LIN {X 0,Y 355.069,Z 437.822,A -85,B 0,C 180,E1 -13382.962,E2 -13382.962} C_VEL
LIN {X 0,Y 354.55,Z 443.957,A -85,B 0,C 180,E1 -13386.644,E2 -13386.644} C_VEL
LIN {X 0,Y 354.327,Z 447.213,A -85,B 0,C 180,E1 -13388.544,E2 -13388.544} C_VEL
LIN {X 0,Y 357.927,Z 462.042,A -85,B 0,C 180,E1 -13389.4,E2 -13389.4} C_VEL
LIN {X 0,Y 360.061,Z 473.49,A -85,B 0,C 180,E1 -13390.214,E2 -13390.214} C_VEL
LIN {X 0,Y 361.071,Z 484.49,A -85,B 0,C 180,E1 -13391.12,E2 -13391.12} C_VEL
LIN {X 0,Y 360.323,Z 493.852,A -85,B 0,C 180,E1 -13391.963,E2 -13391.963} C_VEL
LIN {X 0,Y 358.816,Z 505.238,A -85,B 0,C 180,E1 -13393.208,E2 -13393.208} C_VEL
LIN {X 0,Y 357.676,Z 514.692,A -85,B 0,C 180,E1 -13394.514,E2 -13394.514} C_VEL
LIN {X 0,Y 356.51,Z 523.583,A -85,B 0,C 180,E1 -13396.026,E2 -13396.026} C_VEL
LIN {X 0,Y 355.306,Z 531.692,A -85,B 0,C 180,E1 -13397.723,E2 -13397.723} C_VEL
LIN {X 0,Y 354.632,Z 537.229,A -85,B 0,C 180,E1 -13399.148,E2 -13399.148} C_VEL
LIN {X 0,Y 353.992,Z 542.659,A -85,B 0,C 180,E1 -13400.861,E2 -13400.861} C_VEL
LIN {X 0,Y 353.532,Z 546.923,A -85,B 0,C 180,E1 -13402.576,E2 -13402.576} C_VEL
LIN {X 0,Y 353.311,Z 550.14,A -85,B 0,C 180,E1 -13404.292,E2 -13404.292} C_VEL
LIN {X 0,Y 353.267,Z 551.75,A -85,B 0,C 180,E1 -13405.436,E2 -13405.436} C_VEL
LIN {X 0,Y 353.22,Z 552.959,A -85,B 0,C 180,E1 -13406.578,E2 -13406.578} C_VEL
LIN {X 0,Y 353.216,Z 554.108,A -85,B 0,C 180,E1 -13408.86,E2 -13408.86} C_VEL
LIN {X 0,Y 353.263,Z 554.103,A -85,B 0,C 180,E1 -13410,E2 -13410} C_VEL
LIN {X 0,Y 353.222,Z 553.708,A -85,B 0,C 180,E1 -13411.14,E2 -13411.14} C_VEL
LIN {X 0,Y 353.186,Z 552.882,A -85,B 0,C 180,E1 -13412.281,E2 -13412.281} C_VEL
LIN {X 0,Y 353.225,Z 551.643,A -85,B 0,C 180,E1 -13413.422,E2 -13413.422} C_VEL
LIN {X 0,Y 353.253,Z 548.999,A -85,B 0,C 180,E1 -13415.136,E2 -13415.136} C_VEL
LIN {X 0,Y 353.417,Z 545.326,A -85,B 0,C 180,E1 -13416.852,E2 -13416.852} C_VEL
LIN {X 0,Y 353.731,Z 540.524,A -85,B 0,C 180,E1 -13418.569,E2 -13418.569} C_VEL
LIN {X 0,Y 354.312,Z 533.318,A -85,B 0,C 180,E1 -13420.572,E2 -13420.572} C_VEL
LIN {X 0,Y 355.049,Z 525.43,A -85,B 0,C 180,E1 -13422.285,E2 -13422.285} C_VEL
LIN {X 0,Y 355.823,Z 517.369,A -85,B 0,C 180,E1 -13423.71,E2 -13423.71} C_VEL
LIN {X 0,Y 356.72,Z 507.617,A -85,B 0,C 180,E1 -13425.119,E2 -13425.119} C_VEL
LIN {X 0,Y 357.759,Z 496.542,A -85,B 0,C 180,E1 -13426.402,E2 -13426.402} C_VEL
LIN {X 0,Y 358.683,Z 485.774,A -85,B 0,C 180,E1 -13427.385,E2 -13427.385} C_VEL
LIN {X 0,Y 358.573,Z 480.17,A -85,B 0,C 180,E1 -13427.833,E2 -13427.833} C_VEL
LIN {X 0,Y 357.135,Z 467.764,A -85,B 0,C 180,E1 -13428.691,E2 -13428.691} C_VEL
LIN {X 0,Y 355.076,Z 454.636,A -85,B 0,C 180,E1 -13429.383,E2 -13429.383} C_VEL
LIN {X 0,Y 353.874,Z 447.574,A -85,B 0,C 180,E1 -13429.689,E2 -13429.689} C_VEL
LIN {X 0,Y 354.228,Z 442.075,A -85,B 0,C 180,E1 -13432.76,E2 -13432.76} C_VEL
LIN {X 0,Y 354.602,Z 436.609,A -85,B 0,C 180,E1 -13435.85,E2 -13435.85} C_VEL
LIN {X 0,Y 355.244,Z 428.947,A -85,B 0,C 180,E1 -13440.296,E2 -13440.296} C_VEL
LIN {X 0,Y 355.742,Z 423.445,A -85,B 0,C 180,E1 -13443.583,E2 -13443.583} C_VEL
LIN {X 0,Y 355.998,Z 419.022,A -85,B 0,C 180,E1 -13446.316,E2 -13446.316} C_VEL
LIN {X 0,Y 355.661,Z 415.659,A -85,B 0,C 180,E1 -13448.494,E2 -13448.494} C_VEL
LIN {X 0,Y 354.899,Z 411.28,A -85,B 0,C 180,E1 -13451.56,E2 -13451.56} C_VEL
LIN {X 0,Y 354.812,Z 411.288,A -85,B 0,C 180,E1 -13455.484,E2 -13455.484} C_VEL
LIN {X 0,Y 354.785,Z 411.293,A -85,B 0,C 180,E1 -13459.178,E2 -13459.178} C_VEL
LIN {X 0,Y 354.804,Z 411.287,A -85,B 0,C 180,E1 -13462.401,E2 -13462.401} C_VEL
LIN {X 0,Y 354.808,Z 411.291,A -85,B 0,C 180,E1 -13464.94,E2 -13464.94} C_VEL
LIN {X 0,Y 354.788,Z 411.29,A -85,B 0,C 180,E1 -13468.404,E2 -13468.404} C_VEL
LIN {X 0,Y 354.848,Z 411.281,A -85,B 0,C 180,E1 -13471.619,E2 -13471.619} C_VEL
LIN {X 0,Y 354.893,Z 411.276,A -85,B 0,C 180,E1 -13474.172,E2 -13474.172} C_VEL
LIN {X 0,Y 354.828,Z 411.283,A -85,B 0,C 180,E1 -13477.893,E2 -13477.893} C_VEL
LIN {X 0,Y 354.915,Z 411.273,A -85,B 0,C 180,E1 -13481.891,E2 -13481.891} C_VEL
LIN {X 0,Y 354.935,Z 411.271,A -85,B 0,C 180,E1 -13485.981,E2 -13485.981} C_VEL
LIN {X 0,Y 354.97,Z 411.266,A -85,B 0,C 180,E1 -13489.735,E2 -13489.735} C_VEL
LIN {X 0,Y 355.121,Z 411.249,A -85,B 0,C 180,E1 -13492.037,E2 -13492.037} C_VEL
LIN {X 0,Y 355.089,Z 411.256,A -85,B 0,C 180,E1 -13494.32,E2 -13494.32} C_VEL
LIN {X 0,Y 355.239,Z 411.233,A -85,B 0,C 180,E1 -13497.732,E2 -13497.732} C_VEL
LIN {X 0,Y 355.391,Z 411.216,A -85,B 0,C 180,E1 -13500,E2 -13500} C_VEL
LIN {X 0,Y 355.239,Z 411.237,A -85,B 0,C 180,E1 -13502.267,E2 -13502.267} C_VEL
LIN {X 0,Y 355.13,Z 411.247,A -85,B 0,C 180,E1 -13506.819,E2 -13506.819} C_VEL
LIN {X 0,Y 355.008,Z 411.261,A -85,B 0,C 180,E1 -13509.112,E2 -13509.112} C_VEL
LIN {X 0,Y 354.916,Z 411.274,A -85,B 0,C 180,E1 -13512.581,E2 -13512.581} C_VEL
LIN {X 0,Y 354.882,Z 411.282,A -85,B 0,C 180,E1 -13516.096,E2 -13516.096} C_VEL
LIN {X 0,Y 354.896,Z 411.277,A -85,B 0,C 180,E1 -13518.472,E2 -13518.472} C_VEL
LIN {X 0,Y 354.827,Z 411.288,A -85,B 0,C 180,E1 -13522.106,E2 -13522.106} C_VEL
LIN {X 0,Y 354.892,Z 411.28,A -85,B 0,C 180,E1 -13525.828,E2 -13525.828} C_VEL
LIN {X 0,Y 354.848,Z 411.285,A -85,B 0,C 180,E1 -13529.679,E2 -13529.679} C_VEL
LIN {X 0,Y 354.824,Z 411.289,A -85,B 0,C 180,E1 -13533.683,E2 -13533.683} C_VEL
LIN {X 0,Y 354.796,Z 411.287,A -85,B 0,C 180,E1 -13536.46,E2 -13536.46} C_VEL
LIN {X 0,Y 354.818,Z 411.288,A -85,B 0,C 180,E1 -13539.424,E2 -13539.424} C_VEL
LIN {X 0,Y 354.837,Z 411.282,A -85,B 0,C 180,E1 -13542.877,E2 -13542.877} C_VEL
LIN {X 0,Y 354.861,Z 411.28,A -85,B 0,C 180,E1 -13546.12,E2 -13546.12} C_VEL
LIN {X 0,Y 354.852,Z 411.283,A -85,B 0,C 180,E1 -13549.189,E2 -13549.189} C_VEL
LIN {X 0,Y 354.806,Z 411.285,A -85,B 0,C 180,E1 -13552.403,E2 -13552.403} C_VEL
LIN {X 0,Y 354.809,Z 411.287,A -85,B 0,C 180,E1 -13554.942,E2 -13554.942} C_VEL
LIN {X 0,Y 354.79,Z 411.288,A -85,B 0,C 180,E1 -13558.406,E2 -13558.406} C_VEL
LIN {X 0,Y 354.849,Z 411.283,A -85,B 0,C 180,E1 -13561.62,E2 -13561.62} C_VEL
LIN {X 0,Y 354.896,Z 411.274,A -85,B 0,C 180,E1 -13564.173,E2 -13564.173} C_VEL
LIN {X 0,Y 354.792,Z 411.289,A -85,B 0,C 180,E1 -13566.661,E2 -13566.661} C_VEL
LIN {X 0,Y 354.679,Z 411.364,A -85,B 0,C 180,E1 -13569.257,E2 -13569.257} C_VEL
LIN {X 0,Y 354.506,Z 415.32,A -85,B 0,C 180,E1 -13572.701,E2 -13572.701} C_VEL
LIN {X 0,Y 354.361,Z 419.603,A -85,B 0,C 180,E1 -13576.363,E2 -13576.363} C_VEL
LIN {X 0,Y 354.088,Z 423.661,A -85,B 0,C 180,E1 -13579.71,E2 -13579.71} C_VEL
LIN {X 0,Y 354.096,Z 427.875,A -85,B 0,C 180,E1 -13583.161,E2 -13583.161} C_VEL
LIN {X 0,Y 353.953,Z 429.544,A -85,B 0,C 180,E1 -13584.446,E2 -13584.446} C_VEL
LIN {X 0,Y 356.736,Z 442.632,A -85,B 0,C 180,E1 -13585.073,E2 -13585.073} C_VEL
LIN {X 0,Y 358.816,Z 454.707,A -85,B 0,C 180,E1 -13585.847,E2 -13585.847} C_VEL
LIN {X 0,Y 359.504,Z 461.1,A -85,B 0,C 180,E1 -13586.328,E2 -13586.328} C_VEL
LIN {X 0,Y 358.588,Z 472.632,A -85,B 0,C 180,E1 -13587.29,E2 -13587.29} C_VEL
LIN {X 0,Y 357.635,Z 483.505,A -85,B 0,C 180,E1 -13588.452,E2 -13588.452} C_VEL
LIN {X 0,Y 356.672,Z 493.088,A -85,B 0,C 180,E1 -13589.718,E2 -13589.718} C_VEL
LIN {X 0,Y 355.798,Z 501.822,A -85,B 0,C 180,E1 -13591.132,E2 -13591.132} C_VEL
LIN {X 0,Y 354.892,Z 510.326,A -85,B 0,C 180,E1 -13592.838,E2 -13592.838} C_VEL
LIN {X 0,Y 354.214,Z 517.147,A -85,B 0,C 180,E1 -13594.552,E2 -13594.552} C_VEL
LIN {X 0,Y 353.84,Z 522.956,A -85,B 0,C 180,E1 -13596.401,E2 -13596.401} C_VEL
LIN {X 0,Y 353.541,Z 526.863,A -85,B 0,C 180,E1 -13597.999,E2 -13597.999} C_VEL
LIN {X 0,Y 353.345,Z 529.138,A -85,B 0,C 180,E1 -13599.156,E2 -13599.156} C_VEL
LIN {X 0,Y 353.202,Z 530.929,A -85,B 0,C 180,E1 -13600.316,E2 -13600.316} C_VEL
LIN {X 0,Y 353.163,Z 532.281,A -85,B 0,C 180,E1 -13601.479,E2 -13601.479} C_VEL
LIN {X 0,Y 353.134,Z 533.337,A -85,B 0,C 180,E1 -13602.79,E2 -13602.79} C_VEL
LIN {X 0,Y 353.028,Z 533.879,A -85,B 0,C 180,E1 -13604.999,E2 -13604.999} C_VEL
LIN {X 0,Y 353.191,Z 532.951,A -85,B 0,C 180,E1 -13607.229,E2 -13607.229} C_VEL
LIN {X 0,Y 353.364,Z 531.684,A -85,B 0,C 180,E1 -13608.555,E2 -13608.555} C_VEL
LIN {X 0,Y 353.729,Z 529.087,A -85,B 0,C 180,E1 -13610.346,E2 -13610.346} C_VEL
LIN {X 0,Y 354.177,Z 525.384,A -85,B 0,C 180,E1 -13612.149,E2 -13612.149} C_VEL
LIN {X 0,Y 354.83,Z 520.648,A -85,B 0,C 180,E1 -13613.893,E2 -13613.893} C_VEL
LIN {X 0,Y 355.718,Z 514.138,A -85,B 0,C 180,E1 -13615.763,E2 -13615.763} C_VEL
LIN {X 0,Y 356.686,Z 507.497,A -85,B 0,C 180,E1 -13617.291,E2 -13617.291} C_VEL
LIN {X 0,Y 357.752,Z 499.676,A -85,B 0,C 180,E1 -13618.77,E2 -13618.77} C_VEL
LIN {X 0,Y 359.127,Z 489.929,A -85,B 0,C 180,E1 -13620.259,E2 -13620.259} C_VEL
LIN {X 0,Y 360.487,Z 478.928,A -85,B 0,C 180,E1 -13621.597,E2 -13621.597} C_VEL
LIN {X 0,Y 361.665,Z 468.228,A -85,B 0,C 180,E1 -13622.632,E2 -13622.632} C_VEL
LIN {X 0,Y 362.126,Z 461.499,A -85,B 0,C 180,E1 -13623.181,E2 -13623.181} C_VEL
LIN {X 0,Y 359.869,Z 449.843,A -85,B 0,C 180,E1 -13624.152,E2 -13624.152} C_VEL
LIN {X 0,Y 356.437,Z 437.583,A -85,B 0,C 180,E1 -13625.027,E2 -13625.027} C_VEL
LIN {X 0,Y 353.983,Z 429.889,A -85,B 0,C 180,E1 -13625.51,E2 -13625.51} C_VEL
LIN {X 0,Y 354.281,Z 425.752,A -85,B 0,C 180,E1 -13629.109,E2 -13629.109} C_VEL
LIN {X 0,Y 353.723,Z 424.789,A -85,B 0,C 180,E1 -13630.046,E2 -13630.046} C_VEL
LIN {X 0,Y 350.983,Z 423.48,A -85,B 0,C 180,E1 -13631.58,E2 -13631.58} C_VEL
LIN {X 0,Y 348.634,Z 422.481,A -85,B 0,C 180,E1 -13632.822,E2 -13632.822} C_VEL
LIN {X 0,Y 347.655,Z 421.607,A -85,B 0,C 180,E1 -13633.779,E2 -13633.779} C_VEL
LIN {X 0,Y 347.595,Z 421.276,A -85,B 0,C 180,E1 -13634.102,E2 -13634.102} C_VEL
LIN {X 0,Y 347.873,Z 418.606,A -85,B 0,C 180,E1 -13636.66,E2 -13636.66} C_VEL
LIN {X 0,Y 348.008,Z 415.552,A -85,B 0,C 180,E1 -13639.742,E2 -13639.742} C_VEL
LIN {X 0,Y 347.833,Z 412.784,A -85,B 0,C 180,E1 -13642.688,E2 -13642.688} C_VEL
LIN {X 0,Y 347.783,Z 412.171,A -85,B 0,C 180,E1 -13644.124,E2 -13644.124} C_VEL
LIN {X 0,Y 347.749,Z 412.172,A -85,B 0,C 180,E1 -13648.082,E2 -13648.082} C_VEL
LIN {X 0,Y 347.802,Z 412.162,A -85,B 0,C 180,E1 -13650.99,E2 -13650.99} C_VEL
LIN {X 0,Y 347.827,Z 412.159,A -85,B 0,C 180,E1 -13653.608,E2 -13653.608} C_VEL
LIN {X 0,Y 347.781,Z 412.164,A -85,B 0,C 180,E1 -13656.162,E2 -13656.162} C_VEL
LIN {X 0,Y 347.806,Z 412.161,A -85,B 0,C 180,E1 -13659.909,E2 -13659.909} C_VEL
LIN {X 0,Y 347.861,Z 412.153,A -85,B 0,C 180,E1 -13662.359,E2 -13662.359} C_VEL
LIN {X 0,Y 347.892,Z 412.147,A -85,B 0,C 180,E1 -13665.971,E2 -13665.971} C_VEL
LIN {X 0,Y 347.923,Z 412.144,A -85,B 0,C 180,E1 -13669.526,E2 -13669.526} C_VEL
LIN {X 0,Y 348.069,Z 412.129,A -85,B 0,C 180,E1 -13671.875,E2 -13671.875} C_VEL
LIN {X 0,Y 348.062,Z 412.129,A -85,B 0,C 180,E1 -13674.206,E2 -13674.206} C_VEL
LIN {X 0,Y 348.203,Z 412.111,A -85,B 0,C 180,E1 -13677.687,E2 -13677.687} C_VEL
LIN {X 0,Y 348.341,Z 412.095,A -85,B 0,C 180,E1 -13680,E2 -13680} C_VEL
LIN {X 0,Y 348.203,Z 412.113,A -85,B 0,C 180,E1 -13682.314,E2 -13682.314} C_VEL
LIN {X 0,Y 348.089,Z 412.122,A -85,B 0,C 180,E1 -13686.958,E2 -13686.958} C_VEL
LIN {X 0,Y 347.928,Z 412.146,A -85,B 0,C 180,E1 -13690.475,E2 -13690.475} C_VEL
LIN {X 0,Y 347.894,Z 412.15,A -85,B 0,C 180,E1 -13694.15,E2 -13694.15} C_VEL
LIN {X 0,Y 347.887,Z 412.153,A -85,B 0,C 180,E1 -13698.291,E2 -13698.291} C_VEL
LIN {X 0,Y 347.785,Z 412.167,A -85,B 0,C 180,E1 -13701.635,E2 -13701.635} C_VEL
LIN {X 0,Y 347.809,Z 412.164,A -85,B 0,C 180,E1 -13705.109,E2 -13705.109} C_VEL
LIN {X 0,Y 347.809,Z 412.164,A -85,B 0,C 180,E1 -13707.694,E2 -13707.694} C_VEL
LIN {X 0,Y 347.761,Z 412.168,A -85,B 0,C 180,E1 -13710.347,E2 -13710.347} C_VEL
LIN {X 0,Y 347.742,Z 412.169,A -85,B 0,C 180,E1 -13714.465,E2 -13714.465} C_VEL
LIN {X 0,Y 347.772,Z 412.158,A -85,B 0,C 180,E1 -13717.989,E2 -13717.989} C_VEL
LIN {X 0,Y 347.749,Z 412.17,A -85,B 0,C 180,E1 -13721.831,E2 -13721.831} C_VEL
LIN {X 0,Y 347.76,Z 412.322,A -85,B 0,C 180,E1 -13723.803,E2 -13723.803} C_VEL
LIN {X 0,Y 348.361,Z 415.62,A -85,B 0,C 180,E1 -13726.692,E2 -13726.692} C_VEL
LIN {X 0,Y 349.056,Z 419.568,A -85,B 0,C 180,E1 -13729.917,E2 -13729.917} C_VEL
LIN {X 0,Y 349.61,Z 424.356,A -85,B 0,C 180,E1 -13733.524,E2 -13733.524} C_VEL
LIN {X 0,Y 349.289,Z 428.522,A -85,B 0,C 180,E1 -13736.405,E2 -13736.405} C_VEL
LIN {X 0,Y 348.599,Z 434.182,A -85,B 0,C 180,E1 -13740.102,E2 -13740.102} C_VEL
LIN {X 0,Y 347.818,Z 440.809,A -85,B 0,C 180,E1 -13744.251,E2 -13744.251} C_VEL
LIN {X 0,Y 347.321,Z 447.037,A -85,B 0,C 180,E1 -13748.016,E2 -13748.016} C_VEL
LIN {X 0,Y 350.748,Z 460.4,A -85,B 0,C 180,E1 -13748.797,E2 -13748.797} C_VEL
LIN {X 0,Y 353.117,Z 472.607,A -85,B 0,C 180,E1 -13749.679,E2 -13749.679} C_VEL
LIN {X 0,Y 354.288,Z 483.47,A -85,B 0,C 180,E1 -13750.594,E2 -13750.594} C_VEL
LIN {X 0,Y 354.153,Z 489.992,A -85,B 0,C 180,E1 -13751.188,E2 -13751.188} C_VEL
LIN {X 0,Y 352.75,Z 500.954,A -85,B 0,C 180,E1 -13752.312,E2 -13752.312} C_VEL
LIN {X 0,Y 351.477,Z 509.868,A -85,B 0,C 180,E1 -13753.445,E2 -13753.445} C_VEL
LIN {X 0,Y 350.311,Z 519.035,A -85,B 0,C 180,E1 -13754.882,E2 -13754.882} C_VEL
LIN {X 0,Y 348.992,Z 527.977,A -85,B 0,C 180,E1 -13756.61,E2 -13756.61} C_VEL
LIN {X 0,Y 347.862,Z 535.203,A -85,B 0,C 180,E1 -13758.344,E2 -13758.344} C_VEL
LIN {X 0,Y 347.143,Z 541.01,A -85,B 0,C 180,E1 -13760.091,E2 -13760.091} C_VEL
LIN {X 0,Y 346.633,Z 545.603,A -85,B 0,C 180,E1 -13761.841,E2 -13761.841} C_VEL
LIN {X 0,Y 346.243,Z 549.837,A -85,B 0,C 180,E1 -13764.044,E2 -13764.044} C_VEL
LIN {X 0,Y 346.167,Z 551.63,A -85,B 0,C 180,E1 -13765.342,E2 -13765.342} C_VEL
LIN {X 0,Y 346.143,Z 552.81,A -85,B 0,C 180,E1 -13766.508,E2 -13766.508} C_VEL
LIN {X 0,Y 346.116,Z 553.913,A -85,B 0,C 180,E1 -13768.836,E2 -13768.836} C_VEL
LIN {X 0,Y 346.166,Z 553.888,A -85,B 0,C 180,E1 -13770,E2 -13770} C_VEL
LIN {X 0,Y 346.123,Z 553.469,A -85,B 0,C 180,E1 -13771.163,E2 -13771.163} C_VEL
LIN {X 0,Y 346.097,Z 552.611,A -85,B 0,C 180,E1 -13772.327,E2 -13772.327} C_VEL
LIN {X 0,Y 346.149,Z 551.353,A -85,B 0,C 180,E1 -13773.492,E2 -13773.492} C_VEL
LIN {X 0,Y 346.167,Z 548.283,A -85,B 0,C 180,E1 -13775.45,E2 -13775.45} C_VEL
LIN {X 0,Y 346.449,Z 543.491,A -85,B 0,C 180,E1 -13777.577,E2 -13777.577} C_VEL
LIN {X 0,Y 346.879,Z 537.209,A -85,B 0,C 180,E1 -13779.622,E2 -13779.622} C_VEL
LIN {X 0,Y 347.455,Z 530.358,A -85,B 0,C 180,E1 -13781.374,E2 -13781.374} C_VEL
LIN {X 0,Y 348.432,Z 521.825,A -85,B 0,C 180,E1 -13783.115,E2 -13783.115} C_VEL
LIN {X 0,Y 349.341,Z 513.023,A -85,B 0,C 180,E1 -13784.564,E2 -13784.564} C_VEL
LIN {X 0,Y 350.126,Z 503.701,A -85,B 0,C 180,E1 -13785.827,E2 -13785.827} C_VEL
LIN {X 0,Y 351.177,Z 492.787,A -85,B 0,C 180,E1 -13787.018,E2 -13787.018} C_VEL
LIN {X 0,Y 351.848,Z 482.92,A -85,B 0,C 180,E1 -13787.884,E2 -13787.884} C_VEL
LIN {X 0,Y 350.499,Z 470.9,A -85,B 0,C 180,E1 -13788.795,E2 -13788.795} C_VEL
LIN {X 0,Y 348.564,Z 457.645,A -85,B 0,C 180,E1 -13789.555,E2 -13789.555} C_VEL
LIN {X 0,Y 346.846,Z 447.401,A -85,B 0,C 180,E1 -13790.019,E2 -13790.019} C_VEL
LIN {X 0,Y 347.206,Z 441.747,A -85,B 0,C 180,E1 -13793.247,E2 -13793.247} C_VEL
LIN {X 0,Y 347.573,Z 436.299,A -85,B 0,C 180,E1 -13796.413,E2 -13796.413} C_VEL
LIN {X 0,Y 348.193,Z 429.725,A -85,B 0,C 180,E1 -13800.304,E2 -13800.304} C_VEL
LIN {X 0,Y 348.598,Z 425.337,A -85,B 0,C 180,E1 -13802.979,E2 -13802.979} C_VEL
LIN {X 0,Y 348.952,Z 420.922,A -85,B 0,C 180,E1 -13805.736,E2 -13805.736} C_VEL
LIN {X 0,Y 348.719,Z 417.179,A -85,B 0,C 180,E1 -13808.187,E2 -13808.187} C_VEL
LIN {X 0,Y 347.838,Z 412.16,A -85,B 0,C 180,E1 -13811.816,E2 -13811.816} C_VEL
LIN {X 0,Y 347.793,Z 412.164,A -85,B 0,C 180,E1 -13815.011,E2 -13815.011} C_VEL
LIN {X 0,Y 347.747,Z 412.166,A -85,B 0,C 180,E1 -13818.396,E2 -13818.396} C_VEL
LIN {X 0,Y 347.77,Z 412.162,A -85,B 0,C 180,E1 -13822.01,E2 -13822.01} C_VEL
LIN {X 0,Y 347.74,Z 412.167,A -85,B 0,C 180,E1 -13825.535,E2 -13825.535} C_VEL
LIN {X 0,Y 347.759,Z 412.164,A -85,B 0,C 180,E1 -13829.653,E2 -13829.653} C_VEL
LIN {X 0,Y 347.847,Z 412.158,A -85,B 0,C 180,E1 -13832.744,E2 -13832.744} C_VEL
LIN {X 0,Y 347.782,Z 412.162,A -85,B 0,C 180,E1 -13836.161,E2 -13836.161} C_VEL
LIN {X 0,Y 347.806,Z 412.158,A -85,B 0,C 180,E1 -13839.909,E2 -13839.909} C_VEL
LIN {X 0,Y 347.859,Z 412.154,A -85,B 0,C 180,E1 -13842.359,E2 -13842.359} C_VEL
LIN {X 0,Y 347.89,Z 412.148,A -85,B 0,C 180,E1 -13845.97,E2 -13845.97} C_VEL
LIN {X 0,Y 347.921,Z 412.143,A -85,B 0,C 180,E1 -13849.525,E2 -13849.525} C_VEL
LIN {X 0,Y 348.103,Z 412.122,A -85,B 0,C 180,E1 -13853.042,E2 -13853.042} C_VEL
LIN {X 0,Y 348.201,Z 412.109,A -85,B 0,C 180,E1 -13857.686,E2 -13857.686} C_VEL
LIN {X 0,Y 348.361,Z 412.091,A -85,B 0,C 180,E1 -13860,E2 -13860} C_VEL
LIN {X 0,Y 348.201,Z 412.114,A -85,B 0,C 180,E1 -13862.313,E2 -13862.313} C_VEL
LIN {X 0,Y 348.098,Z 412.122,A -85,B 0,C 180,E1 -13866.958,E2 -13866.958} C_VEL
LIN {X 0,Y 347.96,Z 412.139,A -85,B 0,C 180,E1 -13869.299,E2 -13869.299} C_VEL
LIN {X 0,Y 347.884,Z 412.148,A -85,B 0,C 180,E1 -13872.839,E2 -13872.839} C_VEL
LIN {X 0,Y 347.832,Z 412.157,A -85,B 0,C 180,E1 -13876.432,E2 -13876.432} C_VEL
LIN {X 0,Y 347.845,Z 412.153,A -85,B 0,C 180,E1 -13878.861,E2 -13878.861} C_VEL
LIN {X 0,Y 347.767,Z 412.163,A -85,B 0,C 180,E1 -13882.58,E2 -13882.58} C_VEL
LIN {X 0,Y 347.805,Z 412.158,A -85,B 0,C 180,E1 -13885.109,E2 -13885.109} C_VEL
LIN {X 0,Y 347.805,Z 412.162,A -85,B 0,C 180,E1 -13887.694,E2 -13887.694} C_VEL
LIN {X 0,Y 347.764,Z 412.164,A -85,B 0,C 180,E1 -13890.346,E2 -13890.346} C_VEL
LIN {X 0,Y 347.742,Z 412.169,A -85,B 0,C 180,E1 -13894.044,E2 -13894.044} C_VEL
LIN {X 0,Y 347.761,Z 412.166,A -85,B 0,C 180,E1 -13897.321,E2 -13897.321} C_VEL
LIN {X 0,Y 347.788,Z 412.161,A -85,B 0,C 180,E1 -13900.289,E2 -13900.289} C_VEL
LIN {X 0,Y 347.814,Z 412.161,A -85,B 0,C 180,E1 -13903.394,E2 -13903.394} C_VEL
LIN {X 0,Y 347.813,Z 412.157,A -85,B 0,C 180,E1 -13906.671,E2 -13906.671} C_VEL
LIN {X 0,Y 347.782,Z 412.161,A -85,B 0,C 180,E1 -13910.166,E2 -13910.166} C_VEL
LIN {X 0,Y 347.786,Z 412.16,A -85,B 0,C 180,E1 -13914.126,E2 -13914.126} C_VEL
LIN {X 0,Y 347.735,Z 412.167,A -85,B 0,C 180,E1 -13918.087,E2 -13918.087} C_VEL
LIN {X 0,Y 347.803,Z 412.161,A -85,B 0,C 180,E1 -13920.991,E2 -13920.991} C_VEL
LIN {X 0,Y 347.829,Z 412.157,A -85,B 0,C 180,E1 -13923.608,E2 -13923.608} C_VEL
LIN {X 0,Y 347.768,Z 412.162,A -85,B 0,C 180,E1 -13926.161,E2 -13926.161} C_VEL
LIN {X 0,Y 347.624,Z 412.286,A -85,B 0,C 180,E1 -13929.281,E2 -13929.281} C_VEL
LIN {X 0,Y 347.473,Z 415.723,A -85,B 0,C 180,E1 -13932.339,E2 -13932.339} C_VEL
LIN {X 0,Y 347.303,Z 420.221,A -85,B 0,C 180,E1 -13936.246,E2 -13936.246} C_VEL
LIN {X 0,Y 347.002,Z 425.498,A -85,B 0,C 180,E1 -13940.676,E2 -13940.676} C_VEL
LIN {X 0,Y 346.978,Z 429.068,A -85,B 0,C 180,E1 -13943.604,E2 -13943.604} C_VEL
LIN {X 0,Y 346.92,Z 429.764,A -85,B 0,C 180,E1 -13944.114,E2 -13944.114} C_VEL
LIN {X 0,Y 349.778,Z 443.169,A -85,B 0,C 180,E1 -13944.777,E2 -13944.777} C_VEL
LIN {X 0,Y 351.789,Z 455.127,A -85,B 0,C 180,E1 -13945.56,E2 -13945.56} C_VEL
LIN {X 0,Y 352.642,Z 460.723,A -85,B 0,C 180,E1 -13946,E2 -13946} C_VEL
LIN {X 0,Y 351.729,Z 472.529,A -85,B 0,C 180,E1 -13946.993,E2 -13946.993} C_VEL
LIN {X 0,Y 350.665,Z 484.284,A -85,B 0,C 180,E1 -13948.278,E2 -13948.278} C_VEL
LIN {X 0,Y 349.573,Z 494.739,A -85,B 0,C 180,E1 -13949.712,E2 -13949.712} C_VEL
LIN {X 0,Y 348.675,Z 503.194,A -85,B 0,C 180,E1 -13951.155,E2 -13951.155} C_VEL
LIN {X 0,Y 347.752,Z 511.456,A -85,B 0,C 180,E1 -13952.896,E2 -13952.896} C_VEL
LIN {X 0,Y 347.096,Z 518.107,A -85,B 0,C 180,E1 -13954.646,E2 -13954.646} C_VEL
LIN {X 0,Y 346.75,Z 523.324,A -85,B 0,C 180,E1 -13956.373,E2 -13956.373} C_VEL
LIN {X 0,Y 346.439,Z 527.536,A -85,B 0,C 180,E1 -13958.164,E2 -13958.164} C_VEL
LIN {X 0,Y 346.222,Z 529.707,A -85,B 0,C 180,E1 -13959.346,E2 -13959.346} C_VEL
LIN {X 0,Y 346.098,Z 531.409,A -85,B 0,C 180,E1 -13960.53,E2 -13960.53} C_VEL
LIN {X 0,Y 346.05,Z 532.702,A -85,B 0,C 180,E1 -13961.718,E2 -13961.718} C_VEL
LIN {X 0,Y 346.047,Z 533.587,A -85,B 0,C 180,E1 -13962.909,E2 -13962.909} C_VEL
LIN {X 0,Y 345.951,Z 534.024,A -85,B 0,C 180,E1 -13964.11,E2 -13964.11} C_VEL
LIN {X 0,Y 345.94,Z 534.056,A -85,B 0,C 180,E1 -13965.314,E2 -13965.314} C_VEL
LIN {X 0,Y 346.146,Z 533.135,A -85,B 0,C 180,E1 -13967.395,E2 -13967.395} C_VEL
LIN {X 0,Y 346.331,Z 531.61,A -85,B 0,C 180,E1 -13968.946,E2 -13968.946} C_VEL
LIN {X 0,Y 346.599,Z 529.917,A -85,B 0,C 180,E1 -13970.164,E2 -13970.164} C_VEL
LIN {X 0,Y 347.054,Z 526.46,A -85,B 0,C 180,E1 -13972.001,E2 -13972.001} C_VEL
LIN {X 0,Y 347.735,Z 521.822,A -85,B 0,C 180,E1 -13973.842,E2 -13973.842} C_VEL
LIN {X 0,Y 348.626,Z 515.814,A -85,B 0,C 180,E1 -13975.685,E2 -13975.685} C_VEL
LIN {X 0,Y 349.777,Z 508.192,A -85,B 0,C 180,E1 -13977.525,E2 -13977.525} C_VEL
LIN {X 0,Y 350.932,Z 500.341,A -85,B 0,C 180,E1 -13979.054,E2 -13979.054} C_VEL
LIN {X 0,Y 352.325,Z 490.876,A -85,B 0,C 180,E1 -13980.552,E2 -13980.552} C_VEL
LIN {X 0,Y 353.652,Z 481.234,A -85,B 0,C 180,E1 -13981.777,E2 -13981.777} C_VEL
LIN {X 0,Y 354.812,Z 471.114,A -85,B 0,C 180,E1 -13982.824,E2 -13982.824} C_VEL
LIN {X 0,Y 355.511,Z 462.976,A -85,B 0,C 180,E1 -13983.525,E2 -13983.525} C_VEL
LIN {X 0,Y 353.281,Z 451.251,A -85,B 0,C 180,E1 -13984.55,E2 -13984.55} C_VEL
LIN {X 0,Y 349.669,Z 438.455,A -85,B 0,C 180,E1 -13985.512,E2 -13985.512} C_VEL
LIN {X 0,Y 346.959,Z 430.125,A -85,B 0,C 180,E1 -13986.054,E2 -13986.054} C_VEL
LIN {X 0,Y 347.229,Z 426.626,A -85,B 0,C 180,E1 -13989.145,E2 -13989.145} C_VEL
LIN {X 0,Y 347.496,Z 423.649,A -85,B 0,C 180,E1 -13991.867,E2 -13991.867} C_VEL
LIN {X 0,Y 347.595,Z 421.276,A -85,B 0,C 180,E1 -13994.102,E2 -13994.102} C_VEL
LIN {X 0,Y 347.009,Z 420.369,A -85,B 0,C 180,E1 -13995.059,E2 -13995.059} C_VEL
LIN {X 0,Y 344.308,Z 419.191,A -85,B 0,C 180,E1 -13996.629,E2 -13996.629} C_VEL
LIN {X 0,Y 342.007,Z 418.295,A -85,B 0,C 180,E1 -13997.901,E2 -13997.901} C_VEL
LIN {X 0,Y 341.039,Z 417.498,A -85,B 0,C 180,E1 -13998.879,E2 -13998.879} C_VEL
LIN {X 0,Y 340.971,Z 417.189,A -85,B 0,C 180,E1 -13999.209,E2 -13999.209} C_VEL
LIN {X 0,Y 340.901,Z 414.768,A -85,B 0,C 180,E1 -14001.795,E2 -14001.795} C_VEL
LIN {X 0,Y 340.72,Z 413.212,A -85,B 0,C 180,E1 -14003.556,E2 -14003.556} C_VEL
LIN {X 0,Y 340.691,Z 413.053,A -85,B 0,C 180,E1 -14006.153,E2 -14006.153} C_VEL
LIN {X 0,Y 340.771,Z 413.039,A -85,B 0,C 180,E1 -14010.332,E2 -14010.332} C_VEL
LIN {X 0,Y 340.801,Z 413.036,A -85,B 0,C 180,E1 -14013.02,E2 -14013.02} C_VEL
LIN {X 0,Y 340.75,Z 413.04,A -85,B 0,C 180,E1 -14015.638,E2 -14015.638} C_VEL
LIN {X 0,Y 340.732,Z 413.043,A -85,B 0,C 180,E1 -14019.473,E2 -14019.473} C_VEL
LIN {X 0,Y 340.853,Z 413.027,A -85,B 0,C 180,E1 -14021.984,E2 -14021.984} C_VEL
LIN {X 0,Y 340.864,Z 413.023,A -85,B 0,C 180,E1 -14025.705,E2 -14025.705} C_VEL
LIN {X 0,Y 340.866,Z 413.022,A -85,B 0,C 180,E1 -14029.306,E2 -14029.306} C_VEL
LIN {X 0,Y 341.07,Z 413,A -85,B 0,C 180,E1 -14032.898,E2 -14032.898} C_VEL
LIN {X 0,Y 341.165,Z 412.988,A -85,B 0,C 180,E1 -14037.639,E2 -14037.639} C_VEL
LIN {X 0,Y 341.291,Z 412.973,A -85,B 0,C 180,E1 -14040,E2 -14040} C_VEL
LIN {X 0,Y 341.165,Z 412.99,A -85,B 0,C 180,E1 -14042.361,E2 -14042.361} C_VEL
LIN {X 0,Y 341.057,Z 412.997,A -85,B 0,C 180,E1 -14047.102,E2 -14047.102} C_VEL
LIN {X 0,Y 340.871,Z 413.025,A -85,B 0,C 180,E1 -14050.694,E2 -14050.694} C_VEL
LIN {X 0,Y 340.859,Z 413.028,A -85,B 0,C 180,E1 -14054.325,E2 -14054.325} C_VEL
LIN {X 0,Y 340.834,Z 413.032,A -85,B 0,C 180,E1 -14058.467,E2 -14058.467} C_VEL
LIN {X 0,Y 340.75,Z 413.044,A -85,B 0,C 180,E1 -14061.857,E2 -14061.857} C_VEL
LIN {X 0,Y 340.769,Z 413.039,A -85,B 0,C 180,E1 -14065.665,E2 -14065.665} C_VEL
LIN {X 0,Y 340.739,Z 413.043,A -85,B 0,C 180,E1 -14068.32,E2 -14068.32} C_VEL
LIN {X 0,Y 340.701,Z 413.047,A -85,B 0,C 180,E1 -14071.045,E2 -14071.045} C_VEL
LIN {X 0,Y 340.716,Z 413.043,A -85,B 0,C 180,E1 -14075.279,E2 -14075.279} C_VEL
LIN {X 0,Y 340.708,Z 413.038,A -85,B 0,C 180,E1 -14078.387,E2 -14078.387} C_VEL
LIN {X 0,Y 340.697,Z 413.048,A -85,B 0,C 180,E1 -14082.046,E2 -14082.046} C_VEL
LIN {X 0,Y 340.684,Z 413.071,A -85,B 0,C 180,E1 -14083.132,E2 -14083.132} C_VEL
LIN {X 0,Y 341.267,Z 416.353,A -85,B 0,C 180,E1 -14086.12,E2 -14086.12} C_VEL
LIN {X 0,Y 341.976,Z 420.363,A -85,B 0,C 180,E1 -14089.499,E2 -14089.499} C_VEL
LIN {X 0,Y 342.594,Z 425.029,A -85,B 0,C 180,E1 -14093.135,E2 -14093.135} C_VEL
LIN {X 0,Y 342.481,Z 427.872,A -85,B 0,C 180,E1 -14095.169,E2 -14095.169} C_VEL
LIN {X 0,Y 341.798,Z 433.607,A -85,B 0,C 180,E1 -14099.067,E2 -14099.067} C_VEL
LIN {X 0,Y 340.964,Z 439.751,A -85,B 0,C 180,E1 -14103.034,E2 -14103.034} C_VEL
LIN {X 0,Y 340.487,Z 444.895,A -85,B 0,C 180,E1 -14106.266,E2 -14106.266} C_VEL
LIN {X 0,Y 340.327,Z 446.758,A -85,B 0,C 180,E1 -14107.416,E2 -14107.416} C_VEL
LIN {X 0,Y 344.205,Z 461.861,A -85,B 0,C 180,E1 -14108.374,E2 -14108.374} C_VEL
LIN {X 0,Y 346.604,Z 474.61,A -85,B 0,C 180,E1 -14109.353,E2 -14109.353} C_VEL
LIN {X 0,Y 347.689,Z 485.888,A -85,B 0,C 180,E1 -14110.364,E2 -14110.364} C_VEL
LIN {X 0,Y 346.93,Z 494.898,A -85,B 0,C 180,E1 -14111.241,E2 -14111.241} C_VEL
LIN {X 0,Y 345.298,Z 505.967,A -85,B 0,C 180,E1 -14112.53,E2 -14112.53} C_VEL
LIN {X 0,Y 343.873,Z 516.279,A -85,B 0,C 180,E1 -14114.063,E2 -14114.063} C_VEL
LIN {X 0,Y 342.522,Z 525.398,A -85,B 0,C 180,E1 -14115.746,E2 -14115.746} C_VEL
LIN {X 0,Y 341.244,Z 533.055,A -85,B 0,C 180,E1 -14117.511,E2 -14117.511} C_VEL
LIN {X 0,Y 340.38,Z 539.226,A -85,B 0,C 180,E1 -14119.291,E2 -14119.291} C_VEL
LIN {X 0,Y 339.739,Z 544.149,A -85,B 0,C 180,E1 -14121.075,E2 -14121.075} C_VEL
LIN {X 0,Y 339.321,Z 547.966,A -85,B 0,C 180,E1 -14122.861,E2 -14122.861} C_VEL
LIN {X 0,Y 339.171,Z 549.943,A -85,B 0,C 180,E1 -14124.053,E2 -14124.053} C_VEL
LIN {X 0,Y 339.073,Z 551.512,A -85,B 0,C 180,E1 -14125.244,E2 -14125.244} C_VEL
LIN {X 0,Y 339.068,Z 552.654,A -85,B 0,C 180,E1 -14126.435,E2 -14126.435} C_VEL
LIN {X 0,Y 339.018,Z 553.717,A -85,B 0,C 180,E1 -14128.812,E2 -14128.812} C_VEL
LIN {X 0,Y 339.069,Z 553.674,A -85,B 0,C 180,E1 -14130,E2 -14130} C_VEL
LIN {X 0,Y 339.025,Z 553.223,A -85,B 0,C 180,E1 -14131.188,E2 -14131.188} C_VEL
LIN {X 0,Y 339.074,Z 551.063,A -85,B 0,C 180,E1 -14133.565,E2 -14133.565} C_VEL
LIN {X 0,Y 339.088,Z 549.374,A -85,B 0,C 180,E1 -14134.755,E2 -14134.755} C_VEL
LIN {X 0,Y 339.177,Z 545.964,A -85,B 0,C 180,E1 -14136.544,E2 -14136.544} C_VEL
LIN {X 0,Y 339.513,Z 541.466,A -85,B 0,C 180,E1 -14138.331,E2 -14138.331} C_VEL
LIN {X 0,Y 340.054,Z 534.625,A -85,B 0,C 180,E1 -14140.418,E2 -14140.418} C_VEL
LIN {X 0,Y 340.771,Z 527.17,A -85,B 0,C 180,E1 -14142.204,E2 -14142.204} C_VEL
LIN {X 0,Y 341.585,Z 519.568,A -85,B 0,C 180,E1 -14143.686,E2 -14143.686} C_VEL
LIN {X 0,Y 342.557,Z 510.137,A -85,B 0,C 180,E1 -14145.195,E2 -14145.195} C_VEL
LIN {X 0,Y 343.527,Z 500.087,A -85,B 0,C 180,E1 -14146.49,E2 -14146.49} C_VEL
LIN {X 0,Y 344.663,Z 488.706,A -85,B 0,C 180,E1 -14147.656,E2 -14147.656} C_VEL
LIN {X 0,Y 344.9,Z 483.743,A -85,B 0,C 180,E1 -14148.09,E2 -14148.09} C_VEL
LIN {X 0,Y 343.594,Z 471.597,A -85,B 0,C 180,E1 -14149.048,E2 -14149.048} C_VEL
LIN {X 0,Y 341.71,Z 458.531,A -85,B 0,C 180,E1 -14149.837,E2 -14149.837} C_VEL
LIN {X 0,Y 339.802,Z 447.24,A -85,B 0,C 180,E1 -14150.347,E2 -14150.347} C_VEL
LIN {X 0,Y 340.201,Z 441.419,A -85,B 0,C 180,E1 -14153.755,E2 -14153.755} C_VEL
LIN {X 0,Y 340.578,Z 435.953,A -85,B 0,C 180,E1 -14156.999,E2 -14156.999} C_VEL
LIN {X 0,Y 341.253,Z 429.412,A -85,B 0,C 180,E1 -14160.988,E2 -14160.988} C_VEL
LIN {X 0,Y 341.685,Z 425.002,A -85,B 0,C 180,E1 -14163.734,E2 -14163.734} C_VEL
LIN {X 0,Y 341.923,Z 420.593,A -85,B 0,C 180,E1 -14166.588,E2 -14166.588} C_VEL
LIN {X 0,Y 341.621,Z 417.677,A -85,B 0,C 180,E1 -14168.578,E2 -14168.578} C_VEL
LIN {X 0,Y 340.777,Z 413.039,A -85,B 0,C 180,E1 -14171.963,E2 -14171.963} C_VEL
LIN {X 0,Y 340.701,Z 413.045,A -85,B 0,C 180,E1 -14175.464,E2 -14175.464} C_VEL
LIN {X 0,Y 340.682,Z 413.047,A -85,B 0,C 180,E1 -14178.69,E2 -14178.69} C_VEL
LIN {X 0,Y 340.729,Z 413.039,A -85,B 0,C 180,E1 -14181.772,E2 -14181.772} C_VEL
LIN {X 0,Y 340.718,Z 413.041,A -85,B 0,C 180,E1 -14185.595,E2 -14185.595} C_VEL
LIN {X 0,Y 340.699,Z 413.048,A -85,B 0,C 180,E1 -14188.955,E2 -14188.955} C_VEL
LIN {X 0,Y 340.774,Z 413.036,A -85,B 0,C 180,E1 -14192.473,E2 -14192.473} C_VEL
LIN {X 0,Y 340.75,Z 413.037,A -85,B 0,C 180,E1 -14195.638,E2 -14195.638} C_VEL
LIN {X 0,Y 340.746,Z 413.037,A -85,B 0,C 180,E1 -14199.474,E2 -14199.474} C_VEL
LIN {X 0,Y 340.851,Z 413.025,A -85,B 0,C 180,E1 -14201.984,E2 -14201.984} C_VEL
LIN {X 0,Y 340.862,Z 413.022,A -85,B 0,C 180,E1 -14205.705,E2 -14205.705} C_VEL
LIN {X 0,Y 340.863,Z 413.023,A -85,B 0,C 180,E1 -14209.306,E2 -14209.306} C_VEL
LIN {X 0,Y 341.072,Z 412.998,A -85,B 0,C 180,E1 -14212.898,E2 -14212.898} C_VEL
LIN {X 0,Y 341.163,Z 412.985,A -85,B 0,C 180,E1 -14217.639,E2 -14217.639} C_VEL
LIN {X 0,Y 341.31,Z 412.969,A -85,B 0,C 180,E1 -14220,E2 -14220} C_VEL
LIN {X 0,Y 341.163,Z 412.991,A -85,B 0,C 180,E1 -14222.361,E2 -14222.361} C_VEL
LIN {X 0,Y 341.068,Z 412.997,A -85,B 0,C 180,E1 -14227.102,E2 -14227.102} C_VEL
LIN {X 0,Y 340.865,Z 413.023,A -85,B 0,C 180,E1 -14230.694,E2 -14230.694} C_VEL
LIN {X 0,Y 340.856,Z 413.027,A -85,B 0,C 180,E1 -14234.325,E2 -14234.325} C_VEL
LIN {X 0,Y 340.83,Z 413.028,A -85,B 0,C 180,E1 -14238.467,E2 -14238.467} C_VEL
LIN {X 0,Y 340.747,Z 413.042,A -85,B 0,C 180,E1 -14241.857,E2 -14241.857} C_VEL
LIN {X 0,Y 340.766,Z 413.038,A -85,B 0,C 180,E1 -14245.665,E2 -14245.665} C_VEL
LIN {X 0,Y 340.735,Z 413.04,A -85,B 0,C 180,E1 -14248.32,E2 -14248.32} C_VEL
LIN {X 0,Y 340.709,Z 413.042,A -85,B 0,C 180,E1 -14251.043,E2 -14251.043} C_VEL
LIN {X 0,Y 340.713,Z 413.043,A -85,B 0,C 180,E1 -14255.279,E2 -14255.279} C_VEL
LIN {X 0,Y 340.714,Z 413.041,A -85,B 0,C 180,E1 -14258.389,E2 -14258.389} C_VEL
LIN {X 0,Y 340.72,Z 413.043,A -85,B 0,C 180,E1 -14261.304,E2 -14261.304} C_VEL
LIN {X 0,Y 340.777,Z 413.033,A -85,B 0,C 180,E1 -14264.523,E2 -14264.523} C_VEL
LIN {X 0,Y 340.747,Z 413.039,A -85,B 0,C 180,E1 -14267.945,E2 -14267.945} C_VEL
LIN {X 0,Y 340.73,Z 413.039,A -85,B 0,C 180,E1 -14270.253,E2 -14270.253} C_VEL
LIN {X 0,Y 340.707,Z 413.046,A -85,B 0,C 180,E1 -14273.56,E2 -14273.56} C_VEL
LIN {X 0,Y 340.689,Z 413.044,A -85,B 0,C 180,E1 -14276.154,E2 -14276.154} C_VEL
LIN {X 0,Y 340.772,Z 413.034,A -85,B 0,C 180,E1 -14280.333,E2 -14280.333} C_VEL
LIN {X 0,Y 340.802,Z 413.034,A -85,B 0,C 180,E1 -14283.021,E2 -14283.021} C_VEL
LIN {X 0,Y 340.748,Z 413.039,A -85,B 0,C 180,E1 -14285.639,E2 -14285.639} C_VEL
LIN {X 0,Y 340.588,Z 413.208,A -85,B 0,C 180,E1 -14289.307,E2 -14289.307} C_VEL
LIN {X 0,Y 340.441,Z 416.128,A -85,B 0,C 180,E1 -14291.962,E2 -14291.962} C_VEL
LIN {X 0,Y 340.247,Z 420.841,A -85,B 0,C 180,E1 -14296.123,E2 -14296.123} C_VEL
LIN {X 0,Y 339.996,Z 424.502,A -85,B 0,C 180,E1 -14299.279,E2 -14299.279} C_VEL
LIN {X 0,Y 339.988,Z 428.768,A -85,B 0,C 180,E1 -14302.876,E2 -14302.876} C_VEL
LIN {X 0,Y 339.892,Z 429.834,A -85,B 0,C 180,E1 -14303.753,E2 -14303.753} C_VEL
LIN {X 0,Y 342.946,Z 444.339,A -85,B 0,C 180,E1 -14304.506,E2 -14304.506} C_VEL
LIN {X 0,Y 344.926,Z 456.323,A -85,B 0,C 180,E1 -14305.325,E2 -14305.325} C_VEL
LIN {X 0,Y 345.728,Z 462.412,A -85,B 0,C 180,E1 -14305.821,E2 -14305.821} C_VEL
LIN {X 0,Y 344.764,Z 473.38,A -85,B 0,C 180,E1 -14306.786,E2 -14306.786} C_VEL
LIN {X 0,Y 343.691,Z 485.016,A -85,B 0,C 180,E1 -14308.096,E2 -14308.096} C_VEL
LIN {X 0,Y 342.659,Z 494.422,A -85,B 0,C 180,E1 -14309.413,E2 -14309.413} C_VEL
LIN {X 0,Y 341.74,Z 502.991,A -85,B 0,C 180,E1 -14310.884,E2 -14310.884} C_VEL
LIN {X 0,Y 340.782,Z 511.326,A -85,B 0,C 180,E1 -14312.66,E2 -14312.66} C_VEL
LIN {X 0,Y 340.086,Z 518.041,A -85,B 0,C 180,E1 -14314.445,E2 -14314.445} C_VEL
LIN {X 0,Y 339.793,Z 522.574,A -85,B 0,C 180,E1 -14315.936,E2 -14315.936} C_VEL
LIN {X 0,Y 339.402,Z 526.948,A -85,B 0,C 180,E1 -14317.735,E2 -14317.735} C_VEL
LIN {X 0,Y 339.117,Z 530.247,A -85,B 0,C 180,E1 -14319.543,E2 -14319.543} C_VEL
LIN {X 0,Y 339.002,Z 531.887,A -85,B 0,C 180,E1 -14320.753,E2 -14320.753} C_VEL
LIN {X 0,Y 338.941,Z 533.79,A -85,B 0,C 180,E1 -14322.954,E2 -14322.954} C_VEL
LIN {X 0,Y 338.86,Z 534.262,A -85,B 0,C 180,E1 -14324.411,E2 -14324.411} C_VEL
LIN {X 0,Y 338.855,Z 534.233,A -85,B 0,C 180,E1 -14325.642,E2 -14325.642} C_VEL
LIN {X 0,Y 339.092,Z 533.326,A -85,B 0,C 180,E1 -14327.562,E2 -14327.562} C_VEL
LIN {X 0,Y 339.337,Z 531.543,A -85,B 0,C 180,E1 -14329.352,E2 -14329.352} C_VEL
LIN {X 0,Y 339.832,Z 528.251,A -85,B 0,C 180,E1 -14331.466,E2 -14331.466} C_VEL
LIN {X 0,Y 340.362,Z 524.702,A -85,B 0,C 180,E1 -14333.099,E2 -14333.099} C_VEL
LIN {X 0,Y 341.242,Z 519.354,A -85,B 0,C 180,E1 -14335.015,E2 -14335.015} C_VEL
LIN {X 0,Y 342.258,Z 512.771,A -85,B 0,C 180,E1 -14336.856,E2 -14336.856} C_VEL
LIN {X 0,Y 343.662,Z 504.122,A -85,B 0,C 180,E1 -14338.763,E2 -14338.763} C_VEL
LIN {X 0,Y 344.966,Z 495.566,A -85,B 0,C 180,E1 -14340.28,E2 -14340.28} C_VEL
LIN {X 0,Y 346.381,Z 485.905,A -85,B 0,C 180,E1 -14341.661,E2 -14341.661} C_VEL
LIN {X 0,Y 347.771,Z 475.149,A -85,B 0,C 180,E1 -14342.895,E2 -14342.895} C_VEL
LIN {X 0,Y 348.916,Z 464.648,A -85,B 0,C 180,E1 -14343.858,E2 -14343.858} C_VEL
LIN {X 0,Y 346.937,Z 453.716,A -85,B 0,C 180,E1 -14344.872,E2 -14344.872} C_VEL
LIN {X 0,Y 343.598,Z 441.436,A -85,B 0,C 180,E1 -14345.868,E2 -14345.868} C_VEL
LIN {X 0,Y 339.984,Z 430.319,A -85,B 0,C 180,E1 -14346.634,E2 -14346.634} C_VEL
LIN {X 0,Y 340.285,Z 426.441,A -85,B 0,C 180,E1 -14350.167,E2 -14350.167} C_VEL
LIN {X 0,Y 340.496,Z 423.515,A -85,B 0,C 180,E1 -14352.932,E2 -14352.932} C_VEL
LIN {X 0,Y 340.88,Z 419.214,A -85,B 0,C 180,E1 -14357.128,E2 -14357.128} C_VEL
LIN {X 0,Y 340.971,Z 417.189,A -85,B 0,C 180,E1 -14359.209,E2 -14359.209} C_VEL
LIN {X 0,Y 340.307,Z 416.379,A -85,B 0,C 180,E1 -14360.184,E2 -14360.184} C_VEL
LIN {X 0,Y 337.357,Z 415.377,A -85,B 0,C 180,E1 -14361.774,E2 -14361.774} C_VEL
LIN {X 0,Y 334.834,Z 414.648,A -85,B 0,C 180,E1 -14363.067,E2 -14363.067} C_VEL
LIN {X 0,Y 333.748,Z 414.152,A -85,B 0,C 180,E1 -14364.071,E2 -14364.071} C_VEL
LIN {X 0,Y 333.659,Z 414.062,A -85,B 0,C 180,E1 -14364.413,E2 -14364.413} C_VEL
LIN {X 0,Y 333.638,Z 413.929,A -85,B 0,C 180,E1 -14368.223,E2 -14368.223} C_VEL
LIN {X 0,Y 333.707,Z 413.918,A -85,B 0,C 180,E1 -14371.028,E2 -14371.028} C_VEL
LIN {X 0,Y 333.731,Z 413.915,A -85,B 0,C 180,E1 -14373.754,E2 -14373.754} C_VEL
LIN {X 0,Y 333.652,Z 413.923,A -85,B 0,C 180,E1 -14377.719,E2 -14377.719} C_VEL
LIN {X 0,Y 333.79,Z 413.909,A -85,B 0,C 180,E1 -14381.589,E2 -14381.589} C_VEL
LIN {X 0,Y 333.803,Z 413.903,A -85,B 0,C 180,E1 -14385.577,E2 -14385.577} C_VEL
LIN {X 0,Y 333.829,Z 413.898,A -85,B 0,C 180,E1 -14389.078,E2 -14389.078} C_VEL
LIN {X 0,Y 334.02,Z 413.878,A -85,B 0,C 180,E1 -14392.748,E2 -14392.748} C_VEL
LIN {X 0,Y 333.806,Z 413.906,A -85,B 0,C 180,E1 -14395.169,E2 -14395.169} C_VEL
LIN {X 0,Y 334.102,Z 413.867,A -85,B 0,C 180,E1 -14397.589,E2 -14397.589} C_VEL
LIN {X 0,Y 334.242,Z 413.851,A -85,B 0,C 180,E1 -14400,E2 -14400} C_VEL
LIN {X 0,Y 334.103,Z 413.869,A -85,B 0,C 180,E1 -14402.411,E2 -14402.411} C_VEL
LIN {X 0,Y 334.012,Z 413.879,A -85,B 0,C 180,E1 -14406.039,E2 -14406.039} C_VEL
LIN {X 0,Y 333.98,Z 413.881,A -85,B 0,C 180,E1 -14408.502,E2 -14408.502} C_VEL
LIN {X 0,Y 333.791,Z 413.907,A -85,B 0,C 180,E1 -14412.155,E2 -14412.155} C_VEL
LIN {X 0,Y 333.775,Z 413.911,A -85,B 0,C 180,E1 -14415.887,E2 -14415.887} C_VEL
LIN {X 0,Y 333.793,Z 413.91,A -85,B 0,C 180,E1 -14418.656,E2 -14418.656} C_VEL
LIN {X 0,Y 333.689,Z 413.922,A -85,B 0,C 180,E1 -14422.279,E2 -14422.279} C_VEL
LIN {X 0,Y 333.733,Z 413.918,A -85,B 0,C 180,E1 -14426.247,E2 -14426.247} C_VEL
LIN {X 0,Y 333.708,Z 413.919,A -85,B 0,C 180,E1 -14428.973,E2 -14428.973} C_VEL
LIN {X 0,Y 333.641,Z 413.926,A -85,B 0,C 180,E1 -14432.588,E2 -14432.588} C_VEL
LIN {X 0,Y 333.674,Z 413.919,A -85,B 0,C 180,E1 -14436.14,E2 -14436.14} C_VEL
LIN {X 0,Y 333.645,Z 413.922,A -85,B 0,C 180,E1 -14439.193,E2 -14439.193} C_VEL
LIN {X 0,Y 333.669,Z 414.04,A -85,B 0,C 180,E1 -14442.65,E2 -14442.65} C_VEL
LIN {X 0,Y 334.31,Z 417.7,A -85,B 0,C 180,E1 -14446.074,E2 -14446.074} C_VEL
LIN {X 0,Y 334.989,Z 421.598,A -85,B 0,C 180,E1 -14449.431,E2 -14449.431} C_VEL
LIN {X 0,Y 335.532,Z 425.758,A -85,B 0,C 180,E1 -14452.745,E2 -14452.745} C_VEL
LIN {X 0,Y 335.513,Z 428.483,A -85,B 0,C 180,E1 -14454.78,E2 -14454.78} C_VEL
LIN {X 0,Y 335.109,Z 431.668,A -85,B 0,C 180,E1 -14457.024,E2 -14457.024} C_VEL
LIN {X 0,Y 334.429,Z 436.644,A -85,B 0,C 180,E1 -14460.406,E2 -14460.406} C_VEL
LIN {X 0,Y 333.773,Z 441.764,A -85,B 0,C 180,E1 -14463.757,E2 -14463.757} C_VEL
LIN {X 0,Y 333.337,Z 446.54,A -85,B 0,C 180,E1 -14466.81,E2 -14466.81} C_VEL
LIN {X 0,Y 337.349,Z 461.758,A -85,B 0,C 180,E1 -14467.822,E2 -14467.822} C_VEL
LIN {X 0,Y 339.682,Z 473.873,A -85,B 0,C 180,E1 -14468.78,E2 -14468.78} C_VEL
LIN {X 0,Y 340.892,Z 484.938,A -85,B 0,C 180,E1 -14469.799,E2 -14469.799} C_VEL
LIN {X 0,Y 340.806,Z 491.215,A -85,B 0,C 180,E1 -14470.421,E2 -14470.421} C_VEL
LIN {X 0,Y 339.095,Z 502.947,A -85,B 0,C 180,E1 -14471.731,E2 -14471.731} C_VEL
LIN {X 0,Y 337.636,Z 512.419,A -85,B 0,C 180,E1 -14473.057,E2 -14473.057} C_VEL
LIN {X 0,Y 336.372,Z 521.081,A -85,B 0,C 180,E1 -14474.55,E2 -14474.55} C_VEL
LIN {X 0,Y 334.968,Z 529.547,A -85,B 0,C 180,E1 -14476.347,E2 -14476.347} C_VEL
LIN {X 0,Y 333.784,Z 536.361,A -85,B 0,C 180,E1 -14478.153,E2 -14478.153} C_VEL
LIN {X 0,Y 332.896,Z 542.644,A -85,B 0,C 180,E1 -14480.276,E2 -14480.276} C_VEL
LIN {X 0,Y 332.382,Z 546.766,A -85,B 0,C 180,E1 -14482.1,E2 -14482.1} C_VEL
LIN {X 0,Y 332.067,Z 550.135,A -85,B 0,C 180,E1 -14484.117,E2 -14484.117} C_VEL
LIN {X 0,Y 331.971,Z 552.5,A -85,B 0,C 180,E1 -14486.358,E2 -14486.358} C_VEL
LIN {X 0,Y 331.923,Z 553.523,A -85,B 0,C 180,E1 -14488.787,E2 -14488.787} C_VEL
LIN {X 0,Y 331.972,Z 553.459,A -85,B 0,C 180,E1 -14490,E2 -14490} C_VEL
LIN {X 0,Y 331.93,Z 552.967,A -85,B 0,C 180,E1 -14491.213,E2 -14491.213} C_VEL
LIN {X 0,Y 331.999,Z 550.766,A -85,B 0,C 180,E1 -14493.641,E2 -14493.641} C_VEL
LIN {X 0,Y 332.028,Z 547.368,A -85,B 0,C 180,E1 -14495.818,E2 -14495.818} C_VEL
LIN {X 0,Y 332.327,Z 542.68,A -85,B 0,C 180,E1 -14497.901,E2 -14497.901} C_VEL
LIN {X 0,Y 332.844,Z 536.295,A -85,B 0,C 180,E1 -14500.032,E2 -14500.032} C_VEL
LIN {X 0,Y 333.452,Z 529.323,A -85,B 0,C 180,E1 -14501.858,E2 -14501.858} C_VEL
LIN {X 0,Y 334.487,Z 520.584,A -85,B 0,C 180,E1 -14503.672,E2 -14503.672} C_VEL
LIN {X 0,Y 335.494,Z 511.448,A -85,B 0,C 180,E1 -14505.205,E2 -14505.205} C_VEL
LIN {X 0,Y 336.436,Z 501.729,A -85,B 0,C 180,E1 -14506.536,E2 -14506.536} C_VEL
LIN {X 0,Y 337.545,Z 490.86,A -85,B 0,C 180,E1 -14507.728,E2 -14507.728} C_VEL
LIN {X 0,Y 337.96,Z 484.496,A -85,B 0,C 180,E1 -14508.309,E2 -14508.309} C_VEL
LIN {X 0,Y 336.607,Z 471.636,A -85,B 0,C 180,E1 -14509.358,E2 -14509.358} C_VEL
LIN {X 0,Y 334.747,Z 459.028,A -85,B 0,C 180,E1 -14510.152,E2 -14510.152} C_VEL
LIN {X 0,Y 332.756,Z 447.018,A -85,B 0,C 180,E1 -14510.717,E2 -14510.717} C_VEL
LIN {X 0,Y 333.189,Z 441.09,A -85,B 0,C 180,E1 -14514.279,E2 -14514.279} C_VEL
LIN {X 0,Y 333.594,Z 435.386,A -85,B 0,C 180,E1 -14517.768,E2 -14517.768} C_VEL
LIN {X 0,Y 334.336,Z 429.081,A -85,B 0,C 180,E1 -14521.702,E2 -14521.702} C_VEL
LIN {X 0,Y 334.84,Z 423.881,A -85,B 0,C 180,E1 -14525.057,E2 -14525.057} C_VEL
LIN {X 0,Y 334.799,Z 420.265,A -85,B 0,C 180,E1 -14527.499,E2 -14527.499} C_VEL
LIN {X 0,Y 334.05,Z 415.68,A -85,B 0,C 180,E1 -14530.765,E2 -14530.765} C_VEL
LIN {X 0,Y 333.757,Z 413.914,A -85,B 0,C 180,E1 -14532.158,E2 -14532.158} C_VEL
LIN {X 0,Y 333.631,Z 413.924,A -85,B 0,C 180,E1 -14535.96,E2 -14535.96} C_VEL
LIN {X 0,Y 333.643,Z 413.925,A -85,B 0,C 180,E1 -14539.314,E2 -14539.314} C_VEL
LIN {X 0,Y 333.661,Z 413.924,A -85,B 0,C 180,E1 -14543.167,E2 -14543.167} C_VEL
LIN {X 0,Y 333.669,Z 413.921,A -85,B 0,C 180,E1 -14545.34,E2 -14545.34} C_VEL
LIN {X 0,Y 333.698,Z 413.915,A -85,B 0,C 180,E1 -14549.709,E2 -14549.709} C_VEL
LIN {X 0,Y 333.739,Z 413.911,A -85,B 0,C 180,E1 -14552.4,E2 -14552.4} C_VEL
LIN {X 0,Y 333.721,Z 413.915,A -85,B 0,C 180,E1 -14555.09,E2 -14555.09} C_VEL
LIN {X 0,Y 333.678,Z 413.92,A -85,B 0,C 180,E1 -14559.019,E2 -14559.019} C_VEL
LIN {X 0,Y 333.787,Z 413.903,A -85,B 0,C 180,E1 -14561.589,E2 -14561.589} C_VEL
LIN {X 0,Y 333.801,Z 413.902,A -85,B 0,C 180,E1 -14565.576,E2 -14565.576} C_VEL
LIN {X 0,Y 333.826,Z 413.9,A -85,B 0,C 180,E1 -14569.078,E2 -14569.078} C_VEL
LIN {X 0,Y 334.021,Z 413.878,A -85,B 0,C 180,E1 -14572.747,E2 -14572.747} C_VEL
LIN {X 0,Y 333.808,Z 413.901,A -85,B 0,C 180,E1 -14575.169,E2 -14575.169} C_VEL
LIN {X 0,Y 334.101,Z 413.864,A -85,B 0,C 180,E1 -14577.589,E2 -14577.589} C_VEL
LIN {X 0,Y 334.26,Z 413.847,A -85,B 0,C 180,E1 -14580,E2 -14580} C_VEL
LIN {X 0,Y 334.101,Z 413.87,A -85,B 0,C 180,E1 -14582.411,E2 -14582.411} C_VEL
LIN {X 0,Y 334.018,Z 413.875,A -85,B 0,C 180,E1 -14587.252,E2 -14587.252} C_VEL
LIN {X 0,Y 333.828,Z 413.898,A -85,B 0,C 180,E1 -14590.922,E2 -14590.922} C_VEL
LIN {X 0,Y 333.801,Z 413.903,A -85,B 0,C 180,E1 -14594.634,E2 -14594.634} C_VEL
LIN {X 0,Y 333.789,Z 413.904,A -85,B 0,C 180,E1 -14598.655,E2 -14598.655} C_VEL
LIN {X 0,Y 333.685,Z 413.919,A -85,B 0,C 180,E1 -14602.278,E2 -14602.278} C_VEL
LIN {X 0,Y 333.729,Z 413.914,A -85,B 0,C 180,E1 -14606.247,E2 -14606.247} C_VEL
LIN {X 0,Y 333.705,Z 413.914,A -85,B 0,C 180,E1 -14608.972,E2 -14608.972} C_VEL
LIN {X 0,Y 333.645,Z 413.922,A -85,B 0,C 180,E1 -14612.59,E2 -14612.59} C_VEL
LIN {X 0,Y 333.672,Z 413.92,A -85,B 0,C 180,E1 -14616.139,E2 -14616.139} C_VEL
LIN {X 0,Y 333.679,Z 413.919,A -85,B 0,C 180,E1 -14619.188,E2 -14619.188} C_VEL
LIN {X 0,Y 333.698,Z 413.915,A -85,B 0,C 180,E1 -14622.514,E2 -14622.514} C_VEL
LIN {X 0,Y 333.724,Z 413.914,A -85,B 0,C 180,E1 -14625.978,E2 -14625.978} C_VEL
LIN {X 0,Y 333.698,Z 413.919,A -85,B 0,C 180,E1 -14629.305,E2 -14629.305} C_VEL
LIN {X 0,Y 333.663,Z 413.923,A -85,B 0,C 180,E1 -14633.168,E2 -14633.168} C_VEL
LIN {X 0,Y 333.671,Z 413.924,A -85,B 0,C 180,E1 -14635.342,E2 -14635.342} C_VEL
LIN {X 0,Y 333.7,Z 413.917,A -85,B 0,C 180,E1 -14639.711,E2 -14639.711} C_VEL
LIN {X 0,Y 333.741,Z 413.91,A -85,B 0,C 180,E1 -14642.402,E2 -14642.402} C_VEL
LIN {X 0,Y 333.724,Z 413.916,A -85,B 0,C 180,E1 -14645.091,E2 -14645.091} C_VEL
LIN {X 0,Y 333.565,Z 413.959,A -85,B 0,C 180,E1 -14649.174,E2 -14649.174} C_VEL
LIN {X 0,Y 333.285,Z 417.941,A -85,B 0,C 180,E1 -14652.83,E2 -14652.83} C_VEL
LIN {X 0,Y 333.151,Z 422.151,A -85,B 0,C 180,E1 -14656.583,E2 -14656.583} C_VEL
LIN {X 0,Y 332.873,Z 426.392,A -85,B 0,C 180,E1 -14660.276,E2 -14660.276} C_VEL
LIN {X 0,Y 332.855,Z 430.044,A -85,B 0,C 180,E1 -14663.401,E2 -14663.401} C_VEL
LIN {X 0,Y 335.764,Z 443.534,A -85,B 0,C 180,E1 -14664.106,E2 -14664.106} C_VEL
LIN {X 0,Y 337.919,Z 456.506,A -85,B 0,C 180,E1 -14665.004,E2 -14665.004} C_VEL
LIN {X 0,Y 338.785,Z 464.018,A -85,B 0,C 180,E1 -14665.637,E2 -14665.637} C_VEL
LIN {X 0,Y 337.686,Z 475.653,A -85,B 0,C 180,E1 -14666.719,E2 -14666.719} C_VEL
LIN {X 0,Y 336.593,Z 486.893,A -85,B 0,C 180,E1 -14668.056,E2 -14668.056} C_VEL
LIN {X 0,Y 335.556,Z 495.968,A -85,B 0,C 180,E1 -14669.4,E2 -14669.4} C_VEL
LIN {X 0,Y 334.612,Z 504.28,A -85,B 0,C 180,E1 -14670.903,E2 -14670.903} C_VEL
LIN {X 0,Y 333.637,Z 512.43,A -85,B 0,C 180,E1 -14672.717,E2 -14672.717} C_VEL
LIN {X 0,Y 333.091,Z 517.963,A -85,B 0,C 180,E1 -14674.235,E2 -14674.235} C_VEL
LIN {X 0,Y 332.678,Z 523.368,A -85,B 0,C 180,E1 -14676.063,E2 -14676.063} C_VEL
LIN {X 0,Y 332.294,Z 527.608,A -85,B 0,C 180,E1 -14677.902,E2 -14677.902} C_VEL
LIN {X 0,Y 332.006,Z 530.781,A -85,B 0,C 180,E1 -14679.75,E2 -14679.75} C_VEL
LIN {X 0,Y 331.885,Z 532.362,A -85,B 0,C 180,E1 -14680.987,E2 -14680.987} C_VEL
LIN {X 0,Y 331.845,Z 534.011,A -85,B 0,C 180,E1 -14683.04,E2 -14683.04} C_VEL
LIN {X 0,Y 331.768,Z 534.5,A -85,B 0,C 180,E1 -14684.726,E2 -14684.726} C_VEL
LIN {X 0,Y 331.796,Z 534.4,A -85,B 0,C 180,E1 -14685.983,E2 -14685.983} C_VEL
LIN {X 0,Y 332.023,Z 533.526,A -85,B 0,C 180,E1 -14687.726,E2 -14687.726} C_VEL
LIN {X 0,Y 332.33,Z 531.476,A -85,B 0,C 180,E1 -14689.777,E2 -14689.777} C_VEL
LIN {X 0,Y 332.84,Z 528.444,A -85,B 0,C 180,E1 -14691.71,E2 -14691.71} C_VEL
LIN {X 0,Y 333.499,Z 524.358,A -85,B 0,C 180,E1 -14693.603,E2 -14693.603} C_VEL
LIN {X 0,Y 334.456,Z 518.456,A -85,B 0,C 180,E1 -14695.668,E2 -14695.668} C_VEL
LIN {X 0,Y 335.552,Z 512.035,A -85,B 0,C 180,E1 -14697.437,E2 -14697.437} C_VEL
LIN {X 0,Y 337.015,Z 503.375,A -85,B 0,C 180,E1 -14699.344,E2 -14699.344} C_VEL
LIN {X 0,Y 338.503,Z 494.328,A -85,B 0,C 180,E1 -14700.921,E2 -14700.921} C_VEL
LIN {X 0,Y 340.021,Z 484.603,A -85,B 0,C 180,E1 -14702.29,E2 -14702.29} C_VEL
LIN {X 0,Y 341.508,Z 473.227,A -85,B 0,C 180,E1 -14703.577,E2 -14703.577} C_VEL
LIN {X 0,Y 342.309,Z 466.293,A -85,B 0,C 180,E1 -14704.213,E2 -14704.213} C_VEL
LIN {X 0,Y 340.664,Z 456.551,A -85,B 0,C 180,E1 -14705.168,E2 -14705.168} C_VEL
LIN {X 0,Y 337.623,Z 444.806,A -85,B 0,C 180,E1 -14706.186,E2 -14706.186} C_VEL
LIN {X 0,Y 333.13,Z 431.433,A -85,B 0,C 180,E1 -14707.181,E2 -14707.181} C_VEL
LIN {X 0,Y 332.989,Z 430.53,A -85,B 0,C 180,E1 -14707.258,E2 -14707.258} C_VEL
LIN {X 0,Y 333.304,Z 426.707,A -85,B 0,C 180,E1 -14710.818,E2 -14710.818} C_VEL
LIN {X 0,Y 333.547,Z 423.191,A -85,B 0,C 180,E1 -14714.242,E2 -14714.242} C_VEL
LIN {X 0,Y 333.891,Z 419.786,A -85,B 0,C 180,E1 -14717.658,E2 -14717.658} C_VEL
LIN {X 0,Y 333.931,Z 416.787,A -85,B 0,C 180,E1 -14720.848,E2 -14720.848} C_VEL
LIN {X 0,Y 333.682,Z 414.154,A -85,B 0,C 180,E1 -14723.862,E2 -14723.862} C_VEL
LIN {X 0,Y 333.659,Z 414.062,A -85,B 0,C 180,E1 -14724.413,E2 -14724.413} C_VEL
LIN {X 0,Y 332.988,Z 414.036,A -85,B 0,C 180,E1 -14725.42,E2 -14725.42} C_VEL
LIN {X 0,Y 330.138,Z 414.366,A -85,B 0,C 180,E1 -14727.058,E2 -14727.058} C_VEL
LIN {X 0,Y 327.733,Z 414.665,A -85,B 0,C 180,E1 -14728.386,E2 -14728.386} C_VEL
LIN {X 0,Y 326.711,Z 414.79,A -85,B 0,C 180,E1 -14729.413,E2 -14729.413} C_VEL
LIN {X 0,Y 326.634,Z 414.799,A -85,B 0,C 180,E1 -14729.761,E2 -14729.761} C_VEL
LIN {X 0,Y 326.681,Z 414.794,A -85,B 0,C 180,E1 -14733.142,E2 -14733.142} C_VEL
LIN {X 0,Y 326.644,Z 414.796,A -85,B 0,C 180,E1 -14735.871,E2 -14735.871} C_VEL
LIN {X 0,Y 326.655,Z 414.796,A -85,B 0,C 180,E1 -14739.865,E2 -14739.865} C_VEL
LIN {X 0,Y 326.694,Z 414.79,A -85,B 0,C 180,E1 -14742.472,E2 -14742.472} C_VEL
LIN {X 0,Y 326.754,Z 414.781,A -85,B 0,C 180,E1 -14746.315,E2 -14746.315} C_VEL
LIN {X 0,Y 326.809,Z 414.775,A -85,B 0,C 180,E1 -14750.094,E2 -14750.094} C_VEL
LIN {X 0,Y 326.974,Z 414.756,A -85,B 0,C 180,E1 -14752.59,E2 -14752.59} C_VEL
LIN {X 0,Y 326.773,Z 414.782,A -85,B 0,C 180,E1 -14755.065,E2 -14755.065} C_VEL
LIN {X 0,Y 327.043,Z 414.747,A -85,B 0,C 180,E1 -14757.537,E2 -14757.537} C_VEL
LIN {X 0,Y 327.193,Z 414.729,A -85,B 0,C 180,E1 -14760,E2 -14760} C_VEL
LIN {X 0,Y 327.043,Z 414.748,A -85,B 0,C 180,E1 -14762.463,E2 -14762.463} C_VEL
LIN {X 0,Y 326.987,Z 414.754,A -85,B 0,C 180,E1 -14766.169,E2 -14766.169} C_VEL
LIN {X 0,Y 326.91,Z 414.763,A -85,B 0,C 180,E1 -14768.655,E2 -14768.655} C_VEL
LIN {X 0,Y 326.734,Z 414.786,A -85,B 0,C 180,E1 -14772.422,E2 -14772.422} C_VEL
LIN {X 0,Y 326.75,Z 414.785,A -85,B 0,C 180,E1 -14774.958,E2 -14774.958} C_VEL
LIN {X 0,Y 326.729,Z 414.789,A -85,B 0,C 180,E1 -14778.839,E2 -14778.839} C_VEL
LIN {X 0,Y 326.617,Z 414.803,A -85,B 0,C 180,E1 -14782.788,E2 -14782.788} C_VEL
LIN {X 0,Y 326.687,Z 414.794,A -85,B 0,C 180,E1 -14785.484,E2 -14785.484} C_VEL
LIN {X 0,Y 326.658,Z 414.797,A -85,B 0,C 180,E1 -14789.66,E2 -14789.66} C_VEL
LIN {X 0,Y 326.604,Z 414.802,A -85,B 0,C 180,E1 -14794.02,E2 -14794.02} C_VEL
LIN {X 0,Y 326.626,Z 414.795,A -85,B 0,C 180,E1 -14797.239,E2 -14797.239} C_VEL
LIN {X 0,Y 326.576,Z 414.806,A -85,B 0,C 180,E1 -14801.132,E2 -14801.132} C_VEL
LIN {X 0,Y 326.612,Z 415.017,A -85,B 0,C 180,E1 -14802.139,E2 -14802.139} C_VEL
LIN {X 0,Y 327.157,Z 418.114,A -85,B 0,C 180,E1 -14805.146,E2 -14805.146} C_VEL
LIN {X 0,Y 327.854,Z 421.971,A -85,B 0,C 180,E1 -14808.614,E2 -14808.614} C_VEL
LIN {X 0,Y 328.47,Z 426.478,A -85,B 0,C 180,E1 -14812.341,E2 -14812.341} C_VEL
LIN {X 0,Y 328.506,Z 429.576,A -85,B 0,C 180,E1 -14814.716,E2 -14814.716} C_VEL
LIN {X 0,Y 327.969,Z 433.606,A -85,B 0,C 180,E1 -14817.608,E2 -14817.608} C_VEL
LIN {X 0,Y 327.399,Z 437.661,A -85,B 0,C 180,E1 -14820.415,E2 -14820.415} C_VEL
LIN {X 0,Y 326.618,Z 443.779,A -85,B 0,C 180,E1 -14824.511,E2 -14824.511} C_VEL
LIN {X 0,Y 326.398,Z 446.354,A -85,B 0,C 180,E1 -14826.199,E2 -14826.199} C_VEL
LIN {X 0,Y 328.742,Z 454.819,A -85,B 0,C 180,E1 -14826.742,E2 -14826.742} C_VEL
LIN {X 0,Y 331.408,Z 465.761,A -85,B 0,C 180,E1 -14827.56,E2 -14827.56} C_VEL
LIN {X 0,Y 333.487,Z 478.003,A -85,B 0,C 180,E1 -14828.625,E2 -14828.625} C_VEL
LIN {X 0,Y 334.347,Z 488.799,A -85,B 0,C 180,E1 -14829.707,E2 -14829.707} C_VEL
LIN {X 0,Y 333.373,Z 497.284,A -85,B 0,C 180,E1 -14830.608,E2 -14830.608} C_VEL
LIN {X 0,Y 331.649,Z 507.775,A -85,B 0,C 180,E1 -14831.946,E2 -14831.946} C_VEL
LIN {X 0,Y 330.131,Z 517.622,A -85,B 0,C 180,E1 -14833.526,E2 -14833.526} C_VEL
LIN {X 0,Y 328.779,Z 525.727,A -85,B 0,C 180,E1 -14835.137,E2 -14835.137} C_VEL
LIN {X 0,Y 327.342,Z 533.232,A -85,B 0,C 180,E1 -14836.972,E2 -14836.972} C_VEL
LIN {X 0,Y 326.419,Z 539.287,A -85,B 0,C 180,E1 -14838.827,E2 -14838.827} C_VEL
LIN {X 0,Y 325.674,Z 544.106,A -85,B 0,C 180,E1 -14840.686,E2 -14840.686} C_VEL
LIN {X 0,Y 325.198,Z 547.828,A -85,B 0,C 180,E1 -14842.549,E2 -14842.549} C_VEL
LIN {X 0,Y 324.986,Z 550.233,A -85,B 0,C 180,E1 -14844.144,E2 -14844.144} C_VEL
LIN {X 0,Y 324.878,Z 552.346,A -85,B 0,C 180,E1 -14846.279,E2 -14846.279} C_VEL
LIN {X 0,Y 324.832,Z 553.328,A -85,B 0,C 180,E1 -14848.76,E2 -14848.76} C_VEL
LIN {X 0,Y 324.876,Z 553.238,A -85,B 0,C 180,E1 -14850,E2 -14850} C_VEL
LIN {X 0,Y 324.838,Z 552.711,A -85,B 0,C 180,E1 -14851.239,E2 -14851.239} C_VEL
LIN {X 0,Y 324.847,Z 551.788,A -85,B 0,C 180,E1 -14852.48,E2 -14852.48} C_VEL
LIN {X 0,Y 324.904,Z 550.467,A -85,B 0,C 180,E1 -14853.72,E2 -14853.72} C_VEL
LIN {X 0,Y 324.925,Z 547.364,A -85,B 0,C 180,E1 -14855.751,E2 -14855.751} C_VEL
LIN {X 0,Y 325.149,Z 543.798,A -85,B 0,C 180,E1 -14857.451,E2 -14857.451} C_VEL
LIN {X 0,Y 325.54,Z 538.8,A -85,B 0,C 180,E1 -14859.318,E2 -14859.318} C_VEL
LIN {X 0,Y 326.074,Z 532.5,A -85,B 0,C 180,E1 -14861.185,E2 -14861.185} C_VEL
LIN {X 0,Y 327.006,Z 524.613,A -85,B 0,C 180,E1 -14863.041,E2 -14863.041} C_VEL
LIN {X 0,Y 327.949,Z 516.551,A -85,B 0,C 180,E1 -14864.584,E2 -14864.584} C_VEL
LIN {X 0,Y 328.954,Z 506.689,A -85,B 0,C 180,E1 -14866.125,E2 -14866.125} C_VEL
LIN {X 0,Y 330.135,Z 495.7,A -85,B 0,C 180,E1 -14867.499,E2 -14867.499} C_VEL
LIN {X 0,Y 331.027,Z 486.635,A -85,B 0,C 180,E1 -14868.409,E2 -14868.409} C_VEL
LIN {X 0,Y 330.069,Z 475.978,A -85,B 0,C 180,E1 -14869.354,E2 -14869.354} C_VEL
LIN {X 0,Y 328.394,Z 462.994,A -85,B 0,C 180,E1 -14870.262,E2 -14870.262} C_VEL
LIN {X 0,Y 326.165,Z 449.535,A -85,B 0,C 180,E1 -14870.96,E2 -14870.96} C_VEL
LIN {X 0,Y 325.72,Z 446.81,A -85,B 0,C 180,E1 -14871.103,E2 -14871.103} C_VEL
LIN {X 0,Y 326.207,Z 440.172,A -85,B 0,C 180,E1 -14875.193,E2 -14875.193} C_VEL
LIN {X 0,Y 326.844,Z 433.117,A -85,B 0,C 180,E1 -14879.64,E2 -14879.64} C_VEL
LIN {X 0,Y 327.375,Z 428.738,A -85,B 0,C 180,E1 -14882.458,E2 -14882.458} C_VEL
LIN {X 0,Y 327.84,Z 424.23,A -85,B 0,C 180,E1 -14885.45,E2 -14885.45} C_VEL
LIN {X 0,Y 327.796,Z 421.26,A -85,B 0,C 180,E1 -14887.506,E2 -14887.506} C_VEL
LIN {X 0,Y 326.948,Z 416.207,A -85,B 0,C 180,E1 -14891.205,E2 -14891.205} C_VEL
LIN {X 0,Y 326.69,Z 414.793,A -85,B 0,C 180,E1 -14892.45,E2 -14892.45} C_VEL
LIN {X 0,Y 326.581,Z 414.803,A -85,B 0,C 180,E1 -14896.477,E2 -14896.477} C_VEL
LIN {X 0,Y 326.588,Z 414.801,A -85,B 0,C 180,E1 -14899.79,E2 -14899.79} C_VEL
LIN {X 0,Y 326.626,Z 414.802,A -85,B 0,C 180,E1 -14902.952,E2 -14902.952} C_VEL
LIN {X 0,Y 326.602,Z 414.799,A -85,B 0,C 180,E1 -14905.98,E2 -14905.98} C_VEL
LIN {X 0,Y 326.656,Z 414.793,A -85,B 0,C 180,E1 -14910.34,E2 -14910.34} C_VEL
LIN {X 0,Y 326.684,Z 414.791,A -85,B 0,C 180,E1 -14914.516,E2 -14914.516} C_VEL
LIN {X 0,Y 326.642,Z 414.798,A -85,B 0,C 180,E1 -14918.545,E2 -14918.545} C_VEL
LIN {X 0,Y 326.738,Z 414.782,A -85,B 0,C 180,E1 -14921.177,E2 -14921.177} C_VEL
LIN {X 0,Y 326.756,Z 414.779,A -85,B 0,C 180,E1 -14925.433,E2 -14925.433} C_VEL
LIN {X 0,Y 326.762,Z 414.782,A -85,B 0,C 180,E1 -14928.838,E2 -14928.838} C_VEL
LIN {X 0,Y 326.972,Z 414.757,A -85,B 0,C 180,E1 -14932.59,E2 -14932.59} C_VEL
LIN {X 0,Y 326.775,Z 414.776,A -85,B 0,C 180,E1 -14935.065,E2 -14935.065} C_VEL
LIN {X 0,Y 327.041,Z 414.742,A -85,B 0,C 180,E1 -14937.536,E2 -14937.536} C_VEL
LIN {X 0,Y 327.211,Z 414.724,A -85,B 0,C 180,E1 -14940,E2 -14940} C_VEL
LIN {X 0,Y 327.041,Z 414.748,A -85,B 0,C 180,E1 -14942.463,E2 -14942.463} C_VEL
LIN {X 0,Y 326.964,Z 414.754,A -85,B 0,C 180,E1 -14946.665,E2 -14946.665} C_VEL
LIN {X 0,Y 326.807,Z 414.775,A -85,B 0,C 180,E1 -14949.906,E2 -14949.906} C_VEL
LIN {X 0,Y 326.752,Z 414.78,A -85,B 0,C 180,E1 -14953.685,E2 -14953.685} C_VEL
LIN {X 0,Y 326.692,Z 414.789,A -85,B 0,C 180,E1 -14957.528,E2 -14957.528} C_VEL
LIN {X 0,Y 326.656,Z 414.796,A -85,B 0,C 180,E1 -14960.135,E2 -14960.135} C_VEL
LIN {X 0,Y 326.645,Z 414.797,A -85,B 0,C 180,E1 -14964.129,E2 -14964.129} C_VEL
LIN {X 0,Y 326.679,Z 414.789,A -85,B 0,C 180,E1 -14966.858,E2 -14966.858} C_VEL
LIN {X 0,Y 326.635,Z 414.795,A -85,B 0,C 180,E1 -14970.612,E2 -14970.612} C_VEL
LIN {X 0,Y 326.603,Z 414.802,A -85,B 0,C 180,E1 -14974.02,E2 -14974.02} C_VEL
LIN {X 0,Y 326.625,Z 414.797,A -85,B 0,C 180,E1 -14977.24,E2 -14977.24} C_VEL
LIN {X 0,Y 326.63,Z 414.796,A -85,B 0,C 180,E1 -14980.203,E2 -14980.203} C_VEL
LIN {X 0,Y 326.653,Z 414.798,A -85,B 0,C 180,E1 -14983.51,E2 -14983.51} C_VEL
LIN {X 0,Y 326.646,Z 414.795,A -85,B 0,C 180,E1 -14987.015,E2 -14987.015} C_VEL
LIN {X 0,Y 326.641,Z 414.795,A -85,B 0,C 180,E1 -14990.766,E2 -14990.766} C_VEL
LIN {X 0,Y 326.609,Z 414.798,A -85,B 0,C 180,E1 -14994.481,E2 -14994.481} C_VEL
LIN {X 0,Y 326.605,Z 414.803,A -85,B 0,C 180,E1 -14997.456,E2 -14997.456} C_VEL
LIN {X 0,Y 326.658,Z 414.792,A -85,B 0,C 180,E1 -15000.342,E2 -15000.342} C_VEL
LIN {X 0,Y 326.688,Z 414.789,A -85,B 0,C 180,E1 -15004.517,E2 -15004.517} C_VEL
LIN {X 0,Y 326.522,Z 414.813,A -85,B 0,C 180,E1 -15008.868,E2 -15008.868} C_VEL
LIN {X 0,Y 326.429,Z 415.593,A -85,B 0,C 180,E1 -15009.851,E2 -15009.851} C_VEL
LIN {X 0,Y 326.273,Z 418.369,A -85,B 0,C 180,E1 -15012.449,E2 -15012.449} C_VEL
LIN {X 0,Y 326.114,Z 422.57,A -85,B 0,C 180,E1 -15016.288,E2 -15016.288} C_VEL
LIN {X 0,Y 325.832,Z 426.854,A -85,B 0,C 180,E1 -15020.064,E2 -15020.064} C_VEL
LIN {X 0,Y 325.832,Z 430.333,A -85,B 0,C 180,E1 -15023.038,E2 -15023.038} C_VEL
LIN {X 0,Y 328.661,Z 443.453,A -85,B 0,C 180,E1 -15023.735,E2 -15023.735} C_VEL
LIN {X 0,Y 330.795,Z 455.718,A -85,B 0,C 180,E1 -15024.599,E2 -15024.599} C_VEL
LIN {X 0,Y 331.885,Z 464.6,A -85,B 0,C 180,E1 -15025.36,E2 -15025.36} C_VEL
LIN {X 0,Y 330.762,Z 476.474,A -85,B 0,C 180,E1 -15026.498,E2 -15026.498} C_VEL
LIN {X 0,Y 329.613,Z 487.571,A -85,B 0,C 180,E1 -15027.862,E2 -15027.862} C_VEL
LIN {X 0,Y 328.453,Z 497.459,A -85,B 0,C 180,E1 -15029.387,E2 -15029.387} C_VEL
LIN {X 0,Y 327.5,Z 505.562,A -85,B 0,C 180,E1 -15030.922,E2 -15030.922} C_VEL
LIN {X 0,Y 326.517,Z 513.527,A -85,B 0,C 180,E1 -15032.776,E2 -15032.776} C_VEL
LIN {X 0,Y 325.963,Z 518.903,A -85,B 0,C 180,E1 -15034.328,E2 -15034.328} C_VEL
LIN {X 0,Y 325.546,Z 524.163,A -85,B 0,C 180,E1 -15036.197,E2 -15036.197} C_VEL
LIN {X 0,Y 325.174,Z 528.269,A -85,B 0,C 180,E1 -15038.076,E2 -15038.076} C_VEL
LIN {X 0,Y 324.876,Z 531.317,A -85,B 0,C 180,E1 -15039.966,E2 -15039.966} C_VEL
LIN {X 0,Y 324.784,Z 532.796,A -85,B 0,C 180,E1 -15041.23,E2 -15041.23} C_VEL
LIN {X 0,Y 324.749,Z 534.23,A -85,B 0,C 180,E1 -15043.13,E2 -15043.13} C_VEL
LIN {X 0,Y 324.668,Z 534.733,A -85,B 0,C 180,E1 -15045.056,E2 -15045.056} C_VEL
LIN {X 0,Y 324.735,Z 534.521,A -85,B 0,C 180,E1 -15046.341,E2 -15046.341} C_VEL
LIN {X 0,Y 324.97,Z 533.721,A -85,B 0,C 180,E1 -15047.905,E2 -15047.905} C_VEL
LIN {X 0,Y 325.329,Z 531.367,A -85,B 0,C 180,E1 -15050.221,E2 -15050.221} C_VEL
LIN {X 0,Y 325.817,Z 528.672,A -85,B 0,C 180,E1 -15051.948,E2 -15051.948} C_VEL
LIN {X 0,Y 326.631,Z 523.964,A -85,B 0,C 180,E1 -15054.13,E2 -15054.13} C_VEL
LIN {X 0,Y 327.64,Z 518.312,A -85,B 0,C 180,E1 -15056.112,E2 -15056.112} C_VEL
LIN {X 0,Y 328.928,Z 511.328,A -85,B 0,C 180,E1 -15058.038,E2 -15058.038} C_VEL
LIN {X 0,Y 330.203,Z 504.035,A -85,B 0,C 180,E1 -15059.659,E2 -15059.659} C_VEL
LIN {X 0,Y 331.758,Z 495.125,A -85,B 0,C 180,E1 -15061.265,E2 -15061.265} C_VEL
LIN {X 0,Y 333.39,Z 485.116,A -85,B 0,C 180,E1 -15062.712,E2 -15062.712} C_VEL
LIN {X 0,Y 334.871,Z 474.3,A -85,B 0,C 180,E1 -15063.971,E2 -15063.971} C_VEL
LIN {X 0,Y 335.693,Z 467.169,A -85,B 0,C 180,E1 -15064.657,E2 -15064.657} C_VEL
LIN {X 0,Y 333.633,Z 455.806,A -85,B 0,C 180,E1 -15065.807,E2 -15065.807} C_VEL
LIN {X 0,Y 330.232,Z 443.554,A -85,B 0,C 180,E1 -15066.905,E2 -15066.905} C_VEL
LIN {X 0,Y 325.994,Z 430.743,A -85,B 0,C 180,E1 -15067.889,E2 -15067.889} C_VEL
LIN {X 0,Y 326.34,Z 426.589,A -85,B 0,C 180,E1 -15071.882,E2 -15071.882} C_VEL
LIN {X 0,Y 326.609,Z 423.242,A -85,B 0,C 180,E1 -15075.242,E2 -15075.242} C_VEL
LIN {X 0,Y 326.89,Z 420.382,A -85,B 0,C 180,E1 -15078.204,E2 -15078.204} C_VEL
LIN {X 0,Y 326.906,Z 417.443,A -85,B 0,C 180,E1 -15081.431,E2 -15081.431} C_VEL
LIN {X 0,Y 326.612,Z 414.871,A -85,B 0,C 180,E1 -15084.48,E2 -15084.48} C_VEL
LIN {X 0,Y 326.61,Z 414.805,A -85,B 0,C 180,E1 -15087.456,E2 -15087.456} C_VEL
LIN {X 0,Y 326.634,Z 414.799,A -85,B 0,C 180,E1 -15089.761,E2 -15089.761} C_VEL
LIN {X 0,Y 325.98,Z 414.881,A -85,B 0,C 180,E1 -15090.79,E2 -15090.79} C_VEL
LIN {X 0,Y 323.129,Z 415.235,A -85,B 0,C 180,E1 -15092.464,E2 -15092.464} C_VEL
LIN {X 0,Y 320.709,Z 415.537,A -85,B 0,C 180,E1 -15093.82,E2 -15093.82} C_VEL
LIN {X 0,Y 319.678,Z 415.666,A -85,B 0,C 180,E1 -15094.87,E2 -15094.87} C_VEL
LIN {X 0,Y 319.598,Z 415.676,A -85,B 0,C 180,E1 -15095.226,E2 -15095.226} C_VEL
LIN {X 0,Y 319.599,Z 415.675,A -85,B 0,C 180,E1 -15099.4,E2 -15099.4} C_VEL
LIN {X 0,Y 319.654,Z 415.668,A -85,B 0,C 180,E1 -15102.073,E2 -15102.073} C_VEL
LIN {X 0,Y 319.727,Z 415.655,A -85,B 0,C 180,E1 -15106.008,E2 -15106.008} C_VEL
LIN {X 0,Y 319.753,Z 415.654,A -85,B 0,C 180,E1 -15109.873,E2 -15109.873} C_VEL
LIN {X 0,Y 319.928,Z 415.635,A -85,B 0,C 180,E1 -15112.426,E2 -15112.426} C_VEL
LIN {X 0,Y 319.742,Z 415.658,A -85,B 0,C 180,E1 -15114.956,E2 -15114.956} C_VEL
LIN {X 0,Y 319.986,Z 415.626,A -85,B 0,C 180,E1 -15117.483,E2 -15117.483} C_VEL
LIN {X 0,Y 320.145,Z 415.607,A -85,B 0,C 180,E1 -15120,E2 -15120} C_VEL
LIN {X 0,Y 319.987,Z 415.627,A -85,B 0,C 180,E1 -15122.518,E2 -15122.518} C_VEL
LIN {X 0,Y 319.942,Z 415.631,A -85,B 0,C 180,E1 -15126.306,E2 -15126.306} C_VEL
LIN {X 0,Y 319.839,Z 415.646,A -85,B 0,C 180,E1 -15128.848,E2 -15128.848} C_VEL
LIN {X 0,Y 319.681,Z 415.665,A -85,B 0,C 180,E1 -15132.7,E2 -15132.7} C_VEL
LIN {X 0,Y 319.696,Z 415.663,A -85,B 0,C 180,E1 -15135.296,E2 -15135.296} C_VEL
LIN {X 0,Y 319.671,Z 415.669,A -85,B 0,C 180,E1 -15139.255,E2 -15139.255} C_VEL
LIN {X 0,Y 319.567,Z 415.683,A -85,B 0,C 180,E1 -15143.32,E2 -15143.32} C_VEL
LIN {X 0,Y 319.632,Z 415.674,A -85,B 0,C 180,E1 -15146.089,E2 -15146.089} C_VEL
LIN {X 0,Y 319.587,Z 415.678,A -85,B 0,C 180,E1 -15148.934,E2 -15148.934} C_VEL
LIN {X 0,Y 319.53,Z 415.684,A -85,B 0,C 180,E1 -15151.862,E2 -15151.862} C_VEL
LIN {X 0,Y 319.578,Z 415.676,A -85,B 0,C 180,E1 -15155.544,E2 -15155.544} C_VEL
LIN {X 0,Y 319.557,Z 415.677,A -85,B 0,C 180,E1 -15159.669,E2 -15159.669} C_VEL
LIN {X 0,Y 319.531,Z 415.688,A -85,B 0,C 180,E1 -15161.288,E2 -15161.288} C_VEL
LIN {X 0,Y 320.102,Z 419,A -85,B 0,C 180,E1 -15164.634,E2 -15164.634} C_VEL
LIN {X 0,Y 320.795,Z 422.79,A -85,B 0,C 180,E1 -15168.149,E2 -15168.149} C_VEL
LIN {X 0,Y 321.42,Z 427.188,A -85,B 0,C 180,E1 -15171.921,E2 -15171.921} C_VEL
LIN {X 0,Y 321.537,Z 429.769,A -85,B 0,C 180,E1 -15173.972,E2 -15173.972} C_VEL
LIN {X 0,Y 321.098,Z 433.594,A -85,B 0,C 180,E1 -15176.826,E2 -15176.826} C_VEL
LIN {X 0,Y 320.345,Z 438.652,A -85,B 0,C 180,E1 -15180.421,E2 -15180.421} C_VEL
LIN {X 0,Y 319.586,Z 444.413,A -85,B 0,C 180,E1 -15184.374,E2 -15184.374} C_VEL
LIN {X 0,Y 319.426,Z 446.281,A -85,B 0,C 180,E1 -15185.543,E2 -15185.543} C_VEL
LIN {X 0,Y 322.786,Z 457.993,A -85,B 0,C 180,E1 -15186.353,E2 -15186.353} C_VEL
LIN {X 0,Y 325.275,Z 468.968,A -85,B 0,C 180,E1 -15187.244,E2 -15187.244} C_VEL
LIN {X 0,Y 327.045,Z 480.356,A -85,B 0,C 180,E1 -15188.307,E2 -15188.307} C_VEL
LIN {X 0,Y 327.65,Z 490.978,A -85,B 0,C 180,E1 -15189.437,E2 -15189.437} C_VEL
LIN {X 0,Y 326.272,Z 500.334,A -85,B 0,C 180,E1 -15190.496,E2 -15190.496} C_VEL
LIN {X 0,Y 324.745,Z 509.207,A -85,B 0,C 180,E1 -15191.712,E2 -15191.712} C_VEL
LIN {X 0,Y 323.257,Z 518.323,A -85,B 0,C 180,E1 -15193.255,E2 -15193.255} C_VEL
LIN {X 0,Y 321.657,Z 527.246,A -85,B 0,C 180,E1 -15195.124,E2 -15195.124} C_VEL
LIN {X 0,Y 320.248,Z 534.45,A -85,B 0,C 180,E1 -15197.001,E2 -15197.001} C_VEL
LIN {X 0,Y 319.427,Z 539.332,A -85,B 0,C 180,E1 -15198.579,E2 -15198.579} C_VEL
LIN {X 0,Y 318.649,Z 544.098,A -85,B 0,C 180,E1 -15200.478,E2 -15200.478} C_VEL
LIN {X 0,Y 318.141,Z 547.769,A -85,B 0,C 180,E1 -15202.383,E2 -15202.383} C_VEL
LIN {X 0,Y 317.873,Z 550.376,A -85,B 0,C 180,E1 -15204.229,E2 -15204.229} C_VEL
LIN {X 0,Y 317.788,Z 552.195,A -85,B 0,C 180,E1 -15206.196,E2 -15206.196} C_VEL
LIN {X 0,Y 317.756,Z 552.856,A -85,B 0,C 180,E1 -15207.464,E2 -15207.464} C_VEL
LIN {X 0,Y 317.743,Z 553.134,A -85,B 0,C 180,E1 -15208.732,E2 -15208.732} C_VEL
LIN {X 0,Y 317.784,Z 553.009,A -85,B 0,C 180,E1 -15210,E2 -15210} C_VEL
LIN {X 0,Y 317.75,Z 552.454,A -85,B 0,C 180,E1 -15211.267,E2 -15211.267} C_VEL
LIN {X 0,Y 317.768,Z 551.51,A -85,B 0,C 180,E1 -15212.535,E2 -15212.535} C_VEL
LIN {X 0,Y 317.812,Z 550.167,A -85,B 0,C 180,E1 -15213.804,E2 -15213.804} C_VEL
LIN {X 0,Y 317.846,Z 547.285,A -85,B 0,C 180,E1 -15215.722,E2 -15215.722} C_VEL
LIN {X 0,Y 318.073,Z 543.402,A -85,B 0,C 180,E1 -15217.618,E2 -15217.618} C_VEL
LIN {X 0,Y 318.484,Z 538.351,A -85,B 0,C 180,E1 -15219.526,E2 -15219.526} C_VEL
LIN {X 0,Y 319.059,Z 531.984,A -85,B 0,C 180,E1 -15221.434,E2 -15221.434} C_VEL
LIN {X 0,Y 320.066,Z 524.003,A -85,B 0,C 180,E1 -15223.329,E2 -15223.329} C_VEL
LIN {X 0,Y 321.053,Z 515.855,A -85,B 0,C 180,E1 -15224.904,E2 -15224.904} C_VEL
LIN {X 0,Y 322.084,Z 505.887,A -85,B 0,C 180,E1 -15226.478,E2 -15226.478} C_VEL
LIN {X 0,Y 323.17,Z 496.097,A -85,B 0,C 180,E1 -15227.725,E2 -15227.725} C_VEL
LIN {X 0,Y 324.09,Z 487.135,A -85,B 0,C 180,E1 -15228.654,E2 -15228.654} C_VEL
LIN {X 0,Y 322.986,Z 474.895,A -85,B 0,C 180,E1 -15229.765,E2 -15229.765} C_VEL
LIN {X 0,Y 321.149,Z 461.577,A -85,B 0,C 180,E1 -15230.705,E2 -15230.705} C_VEL
LIN {X 0,Y 318.934,Z 448.456,A -85,B 0,C 180,E1 -15231.389,E2 -15231.389} C_VEL
LIN {X 0,Y 318.662,Z 446.679,A -85,B 0,C 180,E1 -15231.456,E2 -15231.456} C_VEL
LIN {X 0,Y 319.185,Z 440.314,A -85,B 0,C 180,E1 -15235.476,E2 -15235.476} C_VEL
LIN {X 0,Y 319.791,Z 433.87,A -85,B 0,C 180,E1 -15239.634,E2 -15239.634} C_VEL
LIN {X 0,Y 320.336,Z 429.514,A -85,B 0,C 180,E1 -15242.514,E2 -15242.514} C_VEL
LIN {X 0,Y 320.829,Z 424.58,A -85,B 0,C 180,E1 -15245.853,E2 -15245.853} C_VEL
LIN {X 0,Y 320.682,Z 421.712,A -85,B 0,C 180,E1 -15247.91,E2 -15247.91} C_VEL
LIN {X 0,Y 319.833,Z 416.749,A -85,B 0,C 180,E1 -15251.659,E2 -15251.659} C_VEL
LIN {X 0,Y 319.637,Z 415.671,A -85,B 0,C 180,E1 -15252.617,E2 -15252.617} C_VEL
LIN {X 0,Y 319.561,Z 415.678,A -85,B 0,C 180,E1 -15256.53,E2 -15256.53} C_VEL
LIN {X 0,Y 319.543,Z 415.68,A -85,B 0,C 180,E1 -15260.37,E2 -15260.37} C_VEL
LIN {X 0,Y 319.554,Z 415.678,A -85,B 0,C 180,E1 -15263.572,E2 -15263.572} C_VEL
LIN {X 0,Y 319.572,Z 415.678,A -85,B 0,C 180,E1 -15266.686,E2 -15266.686} C_VEL
LIN {X 0,Y 319.586,Z 415.673,A -85,B 0,C 180,E1 -15269.616,E2 -15269.616} C_VEL
LIN {X 0,Y 319.604,Z 415.671,A -85,B 0,C 180,E1 -15272.497,E2 -15272.497} C_VEL
LIN {X 0,Y 319.599,Z 415.672,A -85,B 0,C 180,E1 -15275.303,E2 -15275.303} C_VEL
LIN {X 0,Y 319.592,Z 415.673,A -85,B 0,C 180,E1 -15278.047,E2 -15278.047} C_VEL
LIN {X 0,Y 319.683,Z 415.662,A -85,B 0,C 180,E1 -15280.962,E2 -15280.962} C_VEL
LIN {X 0,Y 319.724,Z 415.655,A -85,B 0,C 180,E1 -15285.276,E2 -15285.276} C_VEL
LIN {X 0,Y 319.75,Z 415.653,A -85,B 0,C 180,E1 -15289.872,E2 -15289.872} C_VEL
LIN {X 0,Y 319.928,Z 415.635,A -85,B 0,C 180,E1 -15292.426,E2 -15292.426} C_VEL
LIN {X 0,Y 319.744,Z 415.652,A -85,B 0,C 180,E1 -15294.956,E2 -15294.956} C_VEL
LIN {X 0,Y 319.985,Z 415.619,A -85,B 0,C 180,E1 -15297.482,E2 -15297.482} C_VEL
LIN {X 0,Y 320.162,Z 415.602,A -85,B 0,C 180,E1 -15300,E2 -15300} C_VEL
LIN {X 0,Y 319.985,Z 415.627,A -85,B 0,C 180,E1 -15302.517,E2 -15302.517} C_VEL
LIN {X 0,Y 319.924,Z 415.632,A -85,B 0,C 180,E1 -15306.656,E2 -15306.656} C_VEL
LIN {X 0,Y 319.751,Z 415.654,A -85,B 0,C 180,E1 -15310.127,E2 -15310.127} C_VEL
LIN {X 0,Y 319.724,Z 415.656,A -85,B 0,C 180,E1 -15314.724,E2 -15314.724} C_VEL
LIN {X 0,Y 319.682,Z 415.661,A -85,B 0,C 180,E1 -15319.038,E2 -15319.038} C_VEL
LIN {X 0,Y 319.563,Z 415.676,A -85,B 0,C 180,E1 -15323.32,E2 -15323.32} C_VEL
LIN {X 0,Y 319.628,Z 415.671,A -85,B 0,C 180,E1 -15326.088,E2 -15326.088} C_VEL
LIN {X 0,Y 319.583,Z 415.672,A -85,B 0,C 180,E1 -15328.934,E2 -15328.934} C_VEL
LIN {X 0,Y 319.532,Z 415.685,A -85,B 0,C 180,E1 -15331.862,E2 -15331.862} C_VEL
LIN {X 0,Y 319.575,Z 415.678,A -85,B 0,C 180,E1 -15335.544,E2 -15335.544} C_VEL
LIN {X 0,Y 319.595,Z 415.674,A -85,B 0,C 180,E1 -15338.005,E2 -15338.005} C_VEL
LIN {X 0,Y 319.597,Z 415.677,A -85,B 0,C 180,E1 -15341.613,E2 -15341.613} C_VEL
LIN {X 0,Y 319.641,Z 415.669,A -85,B 0,C 180,E1 -15345.286,E2 -15345.286} C_VEL
LIN {X 0,Y 319.578,Z 415.674,A -85,B 0,C 180,E1 -15348.721,E2 -15348.721} C_VEL
LIN {X 0,Y 319.595,Z 415.672,A -85,B 0,C 180,E1 -15352.34,E2 -15352.34} C_VEL
LIN {X 0,Y 319.557,Z 415.68,A -85,B 0,C 180,E1 -15355.124,E2 -15355.124} C_VEL
LIN {X 0,Y 319.567,Z 415.679,A -85,B 0,C 180,E1 -15359.059,E2 -15359.059} C_VEL
LIN {X 0,Y 319.606,Z 415.671,A -85,B 0,C 180,E1 -15362.499,E2 -15362.499} C_VEL
LIN {X 0,Y 319.592,Z 415.677,A -85,B 0,C 180,E1 -15365.304,E2 -15365.304} C_VEL
LIN {X 0,Y 319.49,Z 415.747,A -85,B 0,C 180,E1 -15369.141,E2 -15369.141} C_VEL
LIN {X 0,Y 319.249,Z 418.795,A -85,B 0,C 180,E1 -15372.05,E2 -15372.05} C_VEL
LIN {X 0,Y 319.085,Z 422.989,A -85,B 0,C 180,E1 -15375.979,E2 -15375.979} C_VEL
LIN {X 0,Y 318.767,Z 427.27,A -85,B 0,C 180,E1 -15379.842,E2 -15379.842} C_VEL
LIN {X 0,Y 318.781,Z 430.439,A -85,B 0,C 180,E1 -15382.645,E2 -15382.645} C_VEL
LIN {X 0,Y 321.66,Z 443.765,A -85,B 0,C 180,E1 -15383.375,E2 -15383.375} C_VEL
LIN {X 0,Y 323.786,Z 455.712,A -85,B 0,C 180,E1 -15384.239,E2 -15384.239} C_VEL
LIN {X 0,Y 324.989,Z 464.776,A -85,B 0,C 180,E1 -15385.038,E2 -15385.038} C_VEL
LIN {X 0,Y 324.011,Z 475.38,A -85,B 0,C 180,E1 -15386.063,E2 -15386.063} C_VEL
LIN {X 0,Y 322.919,Z 485.979,A -85,B 0,C 180,E1 -15387.35,E2 -15387.35} C_VEL
LIN {X 0,Y 321.79,Z 495.327,A -85,B 0,C 180,E1 -15388.749,E2 -15388.749} C_VEL
LIN {X 0,Y 320.727,Z 503.842,A -85,B 0,C 180,E1 -15390.314,E2 -15390.314} C_VEL
LIN {X 0,Y 319.671,Z 512.136,A -85,B 0,C 180,E1 -15392.205,E2 -15392.205} C_VEL
LIN {X 0,Y 318.963,Z 518.809,A -85,B 0,C 180,E1 -15394.107,E2 -15394.107} C_VEL
LIN {X 0,Y 318.409,Z 524.912,A -85,B 0,C 180,E1 -15396.336,E2 -15396.336} C_VEL
LIN {X 0,Y 318.05,Z 528.886,A -85,B 0,C 180,E1 -15398.258,E2 -15398.258} C_VEL
LIN {X 0,Y 317.75,Z 531.822,A -85,B 0,C 180,E1 -15400.192,E2 -15400.192} C_VEL
LIN {X 0,Y 317.692,Z 533.206,A -85,B 0,C 180,E1 -15401.484,E2 -15401.484} C_VEL
LIN {X 0,Y 317.647,Z 534.445,A -85,B 0,C 180,E1 -15403.218,E2 -15403.218} C_VEL
LIN {X 0,Y 317.603,Z 534.919,A -85,B 0,C 180,E1 -15405.399,E2 -15405.399} C_VEL
LIN {X 0,Y 317.697,Z 534.641,A -85,B 0,C 180,E1 -15406.713,E2 -15406.713} C_VEL
LIN {X 0,Y 317.902,Z 533.926,A -85,B 0,C 180,E1 -15408.081,E2 -15408.081} C_VEL
LIN {X 0,Y 318.073,Z 532.843,A -85,B 0,C 180,E1 -15409.356,E2 -15409.356} C_VEL
LIN {X 0,Y 318.562,Z 530.308,A -85,B 0,C 180,E1 -15411.347,E2 -15411.347} C_VEL
LIN {X 0,Y 319.246,Z 526.677,A -85,B 0,C 180,E1 -15413.344,E2 -15413.344} C_VEL
LIN {X 0,Y 320.143,Z 521.908,A -85,B 0,C 180,E1 -15415.316,E2 -15415.316} C_VEL
LIN {X 0,Y 321.304,Z 515.597,A -85,B 0,C 180,E1 -15417.344,E2 -15417.344} C_VEL
LIN {X 0,Y 322.664,Z 508.783,A -85,B 0,C 180,E1 -15419.088,E2 -15419.088} C_VEL
LIN {X 0,Y 324.324,Z 499.644,A -85,B 0,C 180,E1 -15420.974,E2 -15420.974} C_VEL
LIN {X 0,Y 326.107,Z 489.611,A -85,B 0,C 180,E1 -15422.6,E2 -15422.6} C_VEL
LIN {X 0,Y 327.862,Z 478.358,A -85,B 0,C 180,E1 -15424.056,E2 -15424.056} C_VEL
LIN {X 0,Y 329.068,Z 468.21,A -85,B 0,C 180,E1 -15425.107,E2 -15425.107} C_VEL
LIN {X 0,Y 327.033,Z 456.892,A -85,B 0,C 180,E1 -15426.305,E2 -15426.305} C_VEL
LIN {X 0,Y 323.507,Z 444.339,A -85,B 0,C 180,E1 -15427.482,E2 -15427.482} C_VEL
LIN {X 0,Y 319.589,Z 433.279,A -85,B 0,C 180,E1 -15428.389,E2 -15428.389} C_VEL
LIN {X 0,Y 319.013,Z 430.987,A -85,B 0,C 180,E1 -15428.547,E2 -15428.547} C_VEL
LIN {X 0,Y 319.269,Z 427.926,A -85,B 0,C 180,E1 -15431.545,E2 -15431.545} C_VEL
LIN {X 0,Y 319.586,Z 424.269,A -85,B 0,C 180,E1 -15435.275,E2 -15435.275} C_VEL
LIN {X 0,Y 319.915,Z 420.984,A -85,B 0,C 180,E1 -15438.773,E2 -15438.773} C_VEL
LIN {X 0,Y 319.836,Z 417.905,A -85,B 0,C 180,E1 -15442.283,E2 -15442.283} C_VEL
LIN {X 0,Y 319.557,Z 415.687,A -85,B 0,C 180,E1 -15445.123,E2 -15445.123} C_VEL
LIN {X 0,Y 319.57,Z 415.681,A -85,B 0,C 180,E1 -15449.057,E2 -15449.057} C_VEL
LIN {X 0,Y 319.605,Z 415.674,A -85,B 0,C 180,E1 -15452.498,E2 -15452.498} C_VEL
LIN {X 0,Y 319.598,Z 415.676,A -85,B 0,C 180,E1 -15455.226,E2 -15455.226} C_VEL
LIN {X 0,Y 318.952,Z 415.761,A -85,B 0,C 180,E1 -15456.277,E2 -15456.277} C_VEL
LIN {X 0,Y 316.144,Z 416.11,A -85,B 0,C 180,E1 -15457.99,E2 -15457.99} C_VEL
LIN {X 0,Y 313.75,Z 416.404,A -85,B 0,C 180,E1 -15459.379,E2 -15459.379} C_VEL
LIN {X 0,Y 312.713,Z 416.531,A -85,B 0,C 180,E1 -15460.453,E2 -15460.453} C_VEL
LIN {X 0,Y 312.623,Z 416.542,A -85,B 0,C 180,E1 -15460.816,E2 -15460.816} C_VEL
LIN {X 0,Y 312.695,Z 416.533,A -85,B 0,C 180,E1 -15465.113,E2 -15465.113} C_VEL
LIN {X 0,Y 312.697,Z 416.531,A -85,B 0,C 180,E1 -15469.642,E2 -15469.642} C_VEL
LIN {X 0,Y 312.867,Z 416.515,A -85,B 0,C 180,E1 -15472.254,E2 -15472.254} C_VEL
LIN {X 0,Y 312.713,Z 416.534,A -85,B 0,C 180,E1 -15474.843,E2 -15474.843} C_VEL
LIN {X 0,Y 312.986,Z 416.498,A -85,B 0,C 180,E1 -15478.714,E2 -15478.714} C_VEL
LIN {X 0,Y 312.988,Z 416.499,A -85,B 0,C 180,E1 -15481.287,E2 -15481.287} C_VEL
LIN {X 0,Y 312.713,Z 416.532,A -85,B 0,C 180,E1 -15485.158,E2 -15485.158} C_VEL
LIN {X 0,Y 312.862,Z 416.507,A -85,B 0,C 180,E1 -15487.746,E2 -15487.746} C_VEL
LIN {X 0,Y 312.668,Z 416.539,A -85,B 0,C 180,E1 -15491.672,E2 -15491.672} C_VEL
LIN {X 0,Y 312.696,Z 416.536,A -85,B 0,C 180,E1 -15494.888,E2 -15494.888} C_VEL
LIN {X 0,Y 312.627,Z 416.546,A -85,B 0,C 180,E1 -15499.237,E2 -15499.237} C_VEL
LIN {X 0,Y 312.542,Z 416.557,A -85,B 0,C 180,E1 -15502.79,E2 -15502.79} C_VEL
LIN {X 0,Y 312.6,Z 416.549,A -85,B 0,C 180,E1 -15505.936,E2 -15505.936} C_VEL
LIN {X 0,Y 312.543,Z 416.555,A -85,B 0,C 180,E1 -15509.651,E2 -15509.651} C_VEL
LIN {X 0,Y 312.517,Z 416.557,A -85,B 0,C 180,E1 -15513.689,E2 -15513.689} C_VEL
LIN {X 0,Y 312.518,Z 416.551,A -85,B 0,C 180,E1 -15517.387,E2 -15517.387} C_VEL
LIN {X 0,Y 312.518,Z 416.637,A -85,B 0,C 180,E1 -15520.705,E2 -15520.705} C_VEL
LIN {X 0,Y 313.059,Z 419.891,A -85,B 0,C 180,E1 -15524.102,E2 -15524.102} C_VEL
LIN {X 0,Y 313.757,Z 423.719,A -85,B 0,C 180,E1 -15527.78,E2 -15527.78} C_VEL
LIN {X 0,Y 314.346,Z 427.94,A -85,B 0,C 180,E1 -15531.492,E2 -15531.492} C_VEL
LIN {X 0,Y 314.524,Z 430.426,A -85,B 0,C 180,E1 -15533.554,E2 -15533.554} C_VEL
LIN {X 0,Y 314.093,Z 434.611,A -85,B 0,C 180,E1 -15536.757,E2 -15536.757} C_VEL
LIN {X 0,Y 313.295,Z 439.64,A -85,B 0,C 180,E1 -15540.428,E2 -15540.428} C_VEL
LIN {X 0,Y 312.455,Z 445.924,A -85,B 0,C 180,E1 -15544.83,E2 -15544.83} C_VEL
LIN {X 0,Y 313.328,Z 449.126,A -85,B 0,C 180,E1 -15545.037,E2 -15545.037} C_VEL
LIN {X 0,Y 317.076,Z 462.295,A -85,B 0,C 180,E1 -15546.064,E2 -15546.064} C_VEL
LIN {X 0,Y 319.283,Z 473.378,A -85,B 0,C 180,E1 -15547.048,E2 -15547.048} C_VEL
LIN {X 0,Y 320.7,Z 483.941,A -85,B 0,C 180,E1 -15548.127,E2 -15548.127} C_VEL
LIN {X 0,Y 320.936,Z 493.017,A -85,B 0,C 180,E1 -15549.155,E2 -15549.155} C_VEL
LIN {X 0,Y 319.006,Z 504.31,A -85,B 0,C 180,E1 -15550.536,E2 -15550.536} C_VEL
LIN {X 0,Y 317.337,Z 513.418,A -85,B 0,C 180,E1 -15551.938,E2 -15551.938} C_VEL
LIN {X 0,Y 315.88,Z 521.764,A -85,B 0,C 180,E1 -15553.52,E2 -15553.52} C_VEL
LIN {X 0,Y 314.288,Z 529.95,A -85,B 0,C 180,E1 -15555.43,E2 -15555.43} C_VEL
LIN {X 0,Y 312.887,Z 536.573,A -85,B 0,C 180,E1 -15557.35,E2 -15557.35} C_VEL
LIN {X 0,Y 311.862,Z 542.662,A -85,B 0,C 180,E1 -15559.614,E2 -15559.614} C_VEL
LIN {X 0,Y 311.239,Z 546.639,A -85,B 0,C 180,E1 -15561.56,E2 -15561.56} C_VEL
LIN {X 0,Y 310.892,Z 549.594,A -85,B 0,C 180,E1 -15563.51,E2 -15563.51} C_VEL
LIN {X 0,Y 310.702,Z 552.045,A -85,B 0,C 180,E1 -15566.109,E2 -15566.109} C_VEL
LIN {X 0,Y 310.678,Z 552.685,A -85,B 0,C 180,E1 -15567.407,E2 -15567.407} C_VEL
LIN {X 0,Y 310.657,Z 552.94,A -85,B 0,C 180,E1 -15568.703,E2 -15568.703} C_VEL
LIN {X 0,Y 310.694,Z 552.771,A -85,B 0,C 180,E1 -15570,E2 -15570} C_VEL
LIN {X 0,Y 310.664,Z 552.194,A -85,B 0,C 180,E1 -15571.296,E2 -15571.296} C_VEL
LIN {X 0,Y 310.691,Z 551.227,A -85,B 0,C 180,E1 -15572.593,E2 -15572.593} C_VEL
LIN {X 0,Y 310.722,Z 549.861,A -85,B 0,C 180,E1 -15573.89,E2 -15573.89} C_VEL
LIN {X 0,Y 310.767,Z 547.195,A -85,B 0,C 180,E1 -15575.693,E2 -15575.693} C_VEL
LIN {X 0,Y 311.015,Z 542.998,A -85,B 0,C 180,E1 -15577.792,E2 -15577.792} C_VEL
LIN {X 0,Y 311.544,Z 536.897,A -85,B 0,C 180,E1 -15580.068,E2 -15580.068} C_VEL
LIN {X 0,Y 312.226,Z 530.197,A -85,B 0,C 180,E1 -15582.017,E2 -15582.017} C_VEL
LIN {X 0,Y 313.297,Z 521.878,A -85,B 0,C 180,E1 -15583.954,E2 -15583.954} C_VEL
LIN {X 0,Y 314.485,Z 512.198,A -85,B 0,C 180,E1 -15585.747,E2 -15585.747} C_VEL
LIN {X 0,Y 315.606,Z 501.547,A -85,B 0,C 180,E1 -15587.327,E2 -15587.327} C_VEL
LIN {X 0,Y 316.878,Z 490.811,A -85,B 0,C 180,E1 -15588.591,E2 -15588.591} C_VEL
LIN {X 0,Y 317.034,Z 485.989,A -85,B 0,C 180,E1 -15589.085,E2 -15589.085} C_VEL
LIN {X 0,Y 315.913,Z 474.328,A -85,B 0,C 180,E1 -15590.154,E2 -15590.154} C_VEL
LIN {X 0,Y 314.108,Z 460.702,A -85,B 0,C 180,E1 -15591.126,E2 -15591.126} C_VEL
LIN {X 0,Y 311.727,Z 447.38,A -85,B 0,C 180,E1 -15591.827,E2 -15591.827} C_VEL
LIN {X 0,Y 311.66,Z 446.407,A -85,B 0,C 180,E1 -15591.908,E2 -15591.908} C_VEL
LIN {X 0,Y 312.15,Z 440.459,A -85,B 0,C 180,E1 -15595.763,E2 -15595.763} C_VEL
LIN {X 0,Y 312.857,Z 433.529,A -85,B 0,C 180,E1 -15600.36,E2 -15600.36} C_VEL
LIN {X 0,Y 313.401,Z 429.247,A -85,B 0,C 180,E1 -15603.265,E2 -15603.265} C_VEL
LIN {X 0,Y 313.817,Z 424.951,A -85,B 0,C 180,E1 -15606.27,E2 -15606.27} C_VEL
LIN {X 0,Y 313.46,Z 421.428,A -85,B 0,C 180,E1 -15608.885,E2 -15608.885} C_VEL
LIN {X 0,Y 312.582,Z 416.55,A -85,B 0,C 180,E1 -15612.853,E2 -15612.853} C_VEL
LIN {X 0,Y 312.516,Z 416.555,A -85,B 0,C 180,E1 -15616.022,E2 -15616.022} C_VEL
LIN {X 0,Y 312.5,Z 416.557,A -85,B 0,C 180,E1 -15619.874,E2 -15619.874} C_VEL
LIN {X 0,Y 312.531,Z 416.552,A -85,B 0,C 180,E1 -15624.049,E2 -15624.049} C_VEL
LIN {X 0,Y 312.5,Z 416.558,A -85,B 0,C 180,E1 -15627.333,E2 -15627.333} C_VEL
LIN {X 0,Y 312.547,Z 416.549,A -85,B 0,C 180,E1 -15631.275,E2 -15631.275} C_VEL
LIN {X 0,Y 312.58,Z 416.549,A -85,B 0,C 180,E1 -15634.71,E2 -15634.71} C_VEL
LIN {X 0,Y 312.582,Z 416.546,A -85,B 0,C 180,E1 -15637.528,E2 -15637.528} C_VEL
LIN {X 0,Y 312.632,Z 416.537,A -85,B 0,C 180,E1 -15641.656,E2 -15641.656} C_VEL
LIN {X 0,Y 312.687,Z 416.53,A -85,B 0,C 180,E1 -15645.686,E2 -15645.686} C_VEL
LIN {X 0,Y 312.695,Z 416.531,A -85,B 0,C 180,E1 -15649.641,E2 -15649.641} C_VEL
LIN {X 0,Y 312.868,Z 416.513,A -85,B 0,C 180,E1 -15652.254,E2 -15652.254} C_VEL
LIN {X 0,Y 312.714,Z 416.527,A -85,B 0,C 180,E1 -15654.842,E2 -15654.842} C_VEL
LIN {X 0,Y 312.985,Z 416.495,A -85,B 0,C 180,E1 -15658.713,E2 -15658.713} C_VEL
LIN {X 0,Y 313.114,Z 416.479,A -85,B 0,C 180,E1 -15660,E2 -15660} C_VEL
LIN {X 0,Y 312.932,Z 416.505,A -85,B 0,C 180,E1 -15662.574,E2 -15662.574} C_VEL
LIN {X 0,Y 312.887,Z 416.508,A -85,B 0,C 180,E1 -15666.639,E2 -15666.639} C_VEL
LIN {X 0,Y 312.781,Z 416.518,A -85,B 0,C 180,E1 -15669.049,E2 -15669.049} C_VEL
LIN {X 0,Y 312.628,Z 416.536,A -85,B 0,C 180,E1 -15672.991,E2 -15672.991} C_VEL
LIN {X 0,Y 312.631,Z 416.54,A -85,B 0,C 180,E1 -15675.65,E2 -15675.65} C_VEL
LIN {X 0,Y 312.623,Z 416.541,A -85,B 0,C 180,E1 -15679.236,E2 -15679.236} C_VEL
LIN {X 0,Y 312.539,Z 416.55,A -85,B 0,C 180,E1 -15682.789,E2 -15682.789} C_VEL
LIN {X 0,Y 312.596,Z 416.549,A -85,B 0,C 180,E1 -15685.936,E2 -15685.936} C_VEL
LIN {X 0,Y 312.54,Z 416.553,A -85,B 0,C 180,E1 -15689.65,E2 -15689.65} C_VEL
LIN {X 0,Y 312.514,Z 416.559,A -85,B 0,C 180,E1 -15693.69,E2 -15693.69} C_VEL
LIN {X 0,Y 312.548,Z 416.552,A -85,B 0,C 180,E1 -15697.382,E2 -15697.382} C_VEL
LIN {X 0,Y 312.53,Z 416.552,A -85,B 0,C 180,E1 -15700.703,E2 -15700.703} C_VEL
LIN {X 0,Y 312.59,Z 416.545,A -85,B 0,C 180,E1 -15704.185,E2 -15704.185} C_VEL
LIN {X 0,Y 312.552,Z 416.551,A -85,B 0,C 180,E1 -15707.905,E2 -15707.905} C_VEL
LIN {X 0,Y 312.554,Z 416.551,A -85,B 0,C 180,E1 -15711.906,E2 -15711.906} C_VEL
LIN {X 0,Y 312.503,Z 416.557,A -85,B 0,C 180,E1 -15715.791,E2 -15715.791} C_VEL
LIN {X 0,Y 312.521,Z 416.555,A -85,B 0,C 180,E1 -15718.855,E2 -15718.855} C_VEL
LIN {X 0,Y 312.572,Z 416.548,A -85,B 0,C 180,E1 -15721.825,E2 -15721.825} C_VEL
LIN {X 0,Y 312.579,Z 416.547,A -85,B 0,C 180,E1 -15724.711,E2 -15724.711} C_VEL
LIN {X 0,Y 312.452,Z 416.566,A -85,B 0,C 180,E1 -15728.907,E2 -15728.907} C_VEL
LIN {X 0,Y 312.243,Z 419.211,A -85,B 0,C 180,E1 -15731.633,E2 -15731.633} C_VEL
LIN {X 0,Y 312.039,Z 423.451,A -85,B 0,C 180,E1 -15735.656,E2 -15735.656} C_VEL
LIN {X 0,Y 311.718,Z 427.719,A -85,B 0,C 180,E1 -15739.609,E2 -15739.609} C_VEL
LIN {X 0,Y 311.722,Z 430.605,A -85,B 0,C 180,E1 -15742.226,E2 -15742.226} C_VEL
LIN {X 0,Y 314.867,Z 445.105,A -85,B 0,C 180,E1 -15743.069,E2 -15743.069} C_VEL
LIN {X 0,Y 316.937,Z 456.826,A -85,B 0,C 180,E1 -15743.955,E2 -15743.955} C_VEL
LIN {X 0,Y 318.088,Z 465.913,A -85,B 0,C 180,E1 -15744.791,E2 -15744.791} C_VEL
LIN {X 0,Y 316.956,Z 477.447,A -85,B 0,C 180,E1 -15745.959,E2 -15745.959} C_VEL
LIN {X 0,Y 315.827,Z 487.782,A -85,B 0,C 180,E1 -15747.29,E2 -15747.29} C_VEL
LIN {X 0,Y 314.684,Z 496.813,A -85,B 0,C 180,E1 -15748.721,E2 -15748.721} C_VEL
LIN {X 0,Y 313.623,Z 505.093,A -85,B 0,C 180,E1 -15750.321,E2 -15750.321} C_VEL
LIN {X 0,Y 312.552,Z 513.212,A -85,B 0,C 180,E1 -15752.255,E2 -15752.255} C_VEL
LIN {X 0,Y 311.965,Z 518.713,A -85,B 0,C 180,E1 -15753.875,E2 -15753.875} C_VEL
LIN {X 0,Y 311.449,Z 524.097,A -85,B 0,C 180,E1 -15755.828,E2 -15755.828} C_VEL
LIN {X 0,Y 311.04,Z 528.311,A -85,B 0,C 180,E1 -15757.792,E2 -15757.792} C_VEL
LIN {X 0,Y 310.825,Z 530.545,A -85,B 0,C 180,E1 -15759.107,E2 -15759.107} C_VEL
LIN {X 0,Y 310.63,Z 532.289,A -85,B 0,C 180,E1 -15760.428,E2 -15760.428} C_VEL
LIN {X 0,Y 310.577,Z 533.615,A -85,B 0,C 180,E1 -15761.751,E2 -15761.751} C_VEL
LIN {X 0,Y 310.551,Z 534.659,A -85,B 0,C 180,E1 -15763.315,E2 -15763.315} C_VEL
LIN {X 0,Y 310.517,Z 535.099,A -85,B 0,C 180,E1 -15765.759,E2 -15765.759} C_VEL
LIN {X 0,Y 310.831,Z 534.134,A -85,B 0,C 180,E1 -15768.262,E2 -15768.262} C_VEL
LIN {X 0,Y 311.075,Z 532.785,A -85,B 0,C 180,E1 -15769.809,E2 -15769.809} C_VEL
LIN {X 0,Y 311.61,Z 530.171,A -85,B 0,C 180,E1 -15771.817,E2 -15771.817} C_VEL
LIN {X 0,Y 312.36,Z 526.356,A -85,B 0,C 180,E1 -15773.891,E2 -15773.891} C_VEL
LIN {X 0,Y 313.304,Z 521.796,A -85,B 0,C 180,E1 -15775.775,E2 -15775.775} C_VEL
LIN {X 0,Y 314.678,Z 514.985,A -85,B 0,C 180,E1 -15777.97,E2 -15777.97} C_VEL
LIN {X 0,Y 316.293,Z 507.17,A -85,B 0,C 180,E1 -15779.937,E2 -15779.937} C_VEL
LIN {X 0,Y 317.94,Z 498.558,A -85,B 0,C 180,E1 -15781.667,E2 -15781.667} C_VEL
LIN {X 0,Y 319.825,Z 488.269,A -85,B 0,C 180,E1 -15783.323,E2 -15783.323} C_VEL
LIN {X 0,Y 321.483,Z 478.021,A -85,B 0,C 180,E1 -15784.638,E2 -15784.638} C_VEL
LIN {X 0,Y 322.528,Z 469.968,A -85,B 0,C 180,E1 -15785.488,E2 -15785.488} C_VEL
LIN {X 0,Y 320.585,Z 458.838,A -85,B 0,C 180,E1 -15786.739,E2 -15786.739} C_VEL
LIN {X 0,Y 317.305,Z 446.677,A -85,B 0,C 180,E1 -15787.945,E2 -15787.945} C_VEL
LIN {X 0,Y 312.939,Z 434.127,A -85,B 0,C 180,E1 -15789.035,E2 -15789.035} C_VEL
LIN {X 0,Y 312.037,Z 431.19,A -85,B 0,C 180,E1 -15789.266,E2 -15789.266} C_VEL
LIN {X 0,Y 312.322,Z 428.029,A -85,B 0,C 180,E1 -15792.459,E2 -15792.459} C_VEL
LIN {X 0,Y 312.631,Z 424.677,A -85,B 0,C 180,E1 -15796.001,E2 -15796.001} C_VEL
LIN {X 0,Y 312.894,Z 421.611,A -85,B 0,C 180,E1 -15799.355,E2 -15799.355} C_VEL
LIN {X 0,Y 312.804,Z 418.812,A -85,B 0,C 180,E1 -15802.654,E2 -15802.654} C_VEL
LIN {X 0,Y 312.503,Z 416.565,A -85,B 0,C 180,E1 -15805.79,E2 -15805.79} C_VEL
LIN {X 0,Y 312.523,Z 416.559,A -85,B 0,C 180,E1 -15808.854,E2 -15808.854} C_VEL
LIN {X 0,Y 312.571,Z 416.551,A -85,B 0,C 180,E1 -15811.825,E2 -15811.825} C_VEL
LIN {X 0,Y 312.542,Z 416.552,A -85,B 0,C 180,E1 -15815.213,E2 -15815.213} C_VEL
LIN {X 0,Y 312.533,Z 416.557,A -85,B 0,C 180,E1 -15818.913,E2 -15818.913} C_VEL
LIN {X 0,Y 312.623,Z 416.542,A -85,B 0,C 180,E1 -15820.816,E2 -15820.816} C_VEL
LIN {X 0,Y 311.943,Z 416.629,A -85,B 0,C 180,E1 -15821.892,E2 -15821.892} C_VEL
LIN {X 0,Y 309.09,Z 416.983,A -85,B 0,C 180,E1 -15823.643,E2 -15823.643} C_VEL
LIN {X 0,Y 306.686,Z 417.282,A -85,B 0,C 180,E1 -15825.063,E2 -15825.063} C_VEL
LIN {X 0,Y 305.662,Z 417.407,A -85,B 0,C 180,E1 -15826.162,E2 -15826.162} C_VEL
LIN {X 0,Y 305.582,Z 417.418,A -85,B 0,C 180,E1 -15826.535,E2 -15826.535} C_VEL
LIN {X 0,Y 305.792,Z 417.394,A -85,B 0,C 180,E1 -15831.208,E2 -15831.208} C_VEL
LIN {X 0,Y 305.847,Z 417.388,A -85,B 0,C 180,E1 -15833.403,E2 -15833.403} C_VEL
LIN {X 0,Y 305.952,Z 417.374,A -85,B 0,C 180,E1 -15838.684,E2 -15838.684} C_VEL
LIN {X 0,Y 305.955,Z 417.375,A -85,B 0,C 180,E1 -15841.316,E2 -15841.316} C_VEL
LIN {X 0,Y 305.843,Z 417.386,A -85,B 0,C 180,E1 -15846.598,E2 -15846.598} C_VEL
LIN {X 0,Y 305.732,Z 417.402,A -85,B 0,C 180,E1 -15849.26,E2 -15849.26} C_VEL
LIN {X 0,Y 305.587,Z 417.421,A -85,B 0,C 180,E1 -15853.296,E2 -15853.296} C_VEL
LIN {X 0,Y 305.591,Z 417.422,A -85,B 0,C 180,E1 -15856.021,E2 -15856.021} C_VEL
LIN {X 0,Y 305.573,Z 417.425,A -85,B 0,C 180,E1 -15859.445,E2 -15859.445} C_VEL
LIN {X 0,Y 305.487,Z 417.436,A -85,B 0,C 180,E1 -15863.042,E2 -15863.042} C_VEL
LIN {X 0,Y 305.545,Z 417.429,A -85,B 0,C 180,E1 -15866.228,E2 -15866.228} C_VEL
LIN {X 0,Y 305.493,Z 417.434,A -85,B 0,C 180,E1 -15869.051,E2 -15869.051} C_VEL
LIN {X 0,Y 305.463,Z 417.437,A -85,B 0,C 180,E1 -15873.517,E2 -15873.517} C_VEL
LIN {X 0,Y 305.47,Z 417.431,A -85,B 0,C 180,E1 -15876.74,E2 -15876.74} C_VEL
LIN {X 0,Y 305.498,Z 417.605,A -85,B 0,C 180,E1 -15880.102,E2 -15880.102} C_VEL
LIN {X 0,Y 305.987,Z 420.804,A -85,B 0,C 180,E1 -15883.555,E2 -15883.555} C_VEL
LIN {X 0,Y 306.647,Z 424.446,A -85,B 0,C 180,E1 -15887.173,E2 -15887.173} C_VEL
LIN {X 0,Y 307.148,Z 427.666,A -85,B 0,C 180,E1 -15890.158,E2 -15890.158} C_VEL
LIN {X 0,Y 307.515,Z 431.612,A -85,B 0,C 180,E1 -15893.544,E2 -15893.544} C_VEL
LIN {X 0,Y 307.09,Z 435.608,A -85,B 0,C 180,E1 -15896.684,E2 -15896.684} C_VEL
LIN {X 0,Y 306.174,Z 441.022,A -85,B 0,C 180,E1 -15900.723,E2 -15900.723} C_VEL
LIN {X 0,Y 305.542,Z 445.707,A -85,B 0,C 180,E1 -15904.086,E2 -15904.086} C_VEL
LIN {X 0,Y 306.438,Z 449.004,A -85,B 0,C 180,E1 -15904.312,E2 -15904.312} C_VEL
LIN {X 0,Y 310.208,Z 461.945,A -85,B 0,C 180,E1 -15905.368,E2 -15905.368} C_VEL
LIN {X 0,Y 312.436,Z 472.586,A -85,B 0,C 180,E1 -15906.353,E2 -15906.353} C_VEL
LIN {X 0,Y 314.074,Z 484.786,A -85,B 0,C 180,E1 -15907.641,E2 -15907.641} C_VEL
LIN {X 0,Y 314.347,Z 493.653,A -85,B 0,C 180,E1 -15908.697,E2 -15908.697} C_VEL
LIN {X 0,Y 312.352,Z 504.755,A -85,B 0,C 180,E1 -15910.104,E2 -15910.104} C_VEL
LIN {X 0,Y 310.412,Z 514.847,A -85,B 0,C 180,E1 -15911.734,E2 -15911.734} C_VEL
LIN {X 0,Y 308.802,Z 523.476,A -85,B 0,C 180,E1 -15913.472,E2 -15913.472} C_VEL
LIN {X 0,Y 307.142,Z 531.329,A -85,B 0,C 180,E1 -15915.422,E2 -15915.422} C_VEL
LIN {X 0,Y 305.757,Z 537.628,A -85,B 0,C 180,E1 -15917.387,E2 -15917.387} C_VEL
LIN {X 0,Y 304.845,Z 542.661,A -85,B 0,C 180,E1 -15919.372,E2 -15919.372} C_VEL
LIN {X 0,Y 304.191,Z 546.586,A -85,B 0,C 180,E1 -15921.363,E2 -15921.363} C_VEL
LIN {X 0,Y 303.828,Z 549.501,A -85,B 0,C 180,E1 -15923.358,E2 -15923.358} C_VEL
LIN {X 0,Y 303.599,Z 551.895,A -85,B 0,C 180,E1 -15926.018,E2 -15926.018} C_VEL
LIN {X 0,Y 303.603,Z 552.514,A -85,B 0,C 180,E1 -15927.346,E2 -15927.346} C_VEL
LIN {X 0,Y 303.574,Z 552.738,A -85,B 0,C 180,E1 -15928.673,E2 -15928.673} C_VEL
LIN {X 0,Y 303.606,Z 552.533,A -85,B 0,C 180,E1 -15930,E2 -15930} C_VEL
LIN {X 0,Y 303.58,Z 551.934,A -85,B 0,C 180,E1 -15931.326,E2 -15931.326} C_VEL
LIN {X 0,Y 303.615,Z 550.945,A -85,B 0,C 180,E1 -15932.653,E2 -15932.653} C_VEL
LIN {X 0,Y 303.635,Z 549.547,A -85,B 0,C 180,E1 -15933.981,E2 -15933.981} C_VEL
LIN {X 0,Y 303.661,Z 547.189,A -85,B 0,C 180,E1 -15935.611,E2 -15935.611} C_VEL
LIN {X 0,Y 303.953,Z 542.592,A -85,B 0,C 180,E1 -15937.974,E2 -15937.974} C_VEL
LIN {X 0,Y 304.509,Z 536.409,A -85,B 0,C 180,E1 -15940.303,E2 -15940.303} C_VEL
LIN {X 0,Y 305.223,Z 529.644,A -85,B 0,C 180,E1 -15942.297,E2 -15942.297} C_VEL
LIN {X 0,Y 306.335,Z 521.247,A -85,B 0,C 180,E1 -15944.278,E2 -15944.278} C_VEL
LIN {X 0,Y 307.478,Z 512.582,A -85,B 0,C 180,E1 -15945.919,E2 -15945.919} C_VEL
LIN {X 0,Y 308.639,Z 501.859,A -85,B 0,C 180,E1 -15947.56,E2 -15947.56} C_VEL
LIN {X 0,Y 309.947,Z 491.237,A -85,B 0,C 180,E1 -15948.851,E2 -15948.851} C_VEL
LIN {X 0,Y 310.071,Z 486.466,A -85,B 0,C 180,E1 -15949.358,E2 -15949.358} C_VEL
LIN {X 0,Y 308.875,Z 473.853,A -85,B 0,C 180,E1 -15950.548,E2 -15950.548} C_VEL
LIN {X 0,Y 307.076,Z 460.709,A -85,B 0,C 180,E1 -15951.513,E2 -15951.513} C_VEL
LIN {X 0,Y 304.872,Z 448.079,A -85,B 0,C 180,E1 -15952.207,E2 -15952.207} C_VEL
LIN {X 0,Y 304.604,Z 446.254,A -85,B 0,C 180,E1 -15952.311,E2 -15952.311} C_VEL
LIN {X 0,Y 305.114,Z 440.61,A -85,B 0,C 180,E1 -15956.06,E2 -15956.06} C_VEL
LIN {X 0,Y 305.976,Z 433.188,A -85,B 0,C 180,E1 -15961.107,E2 -15961.107} C_VEL
LIN {X 0,Y 306.677,Z 427.722,A -85,B 0,C 180,E1 -15964.953,E2 -15964.953} C_VEL
LIN {X 0,Y 306.71,Z 424.389,A -85,B 0,C 180,E1 -15967.394,E2 -15967.394} C_VEL
LIN {X 0,Y 306.02,Z 420.137,A -85,B 0,C 180,E1 -15970.723,E2 -15970.723} C_VEL
LIN {X 0,Y 305.533,Z 417.429,A -85,B 0,C 180,E1 -15973.071,E2 -15973.071} C_VEL
LIN {X 0,Y 305.46,Z 417.436,A -85,B 0,C 180,E1 -15977.412,E2 -15977.412} C_VEL
LIN {X 0,Y 305.472,Z 417.433,A -85,B 0,C 180,E1 -15981.597,E2 -15981.597} C_VEL
LIN {X 0,Y 305.458,Z 417.438,A -85,B 0,C 180,E1 -15984.886,E2 -15984.886} C_VEL
LIN {X 0,Y 305.447,Z 417.436,A -85,B 0,C 180,E1 -15988.354,E2 -15988.354} C_VEL
LIN {X 0,Y 305.516,Z 417.425,A -85,B 0,C 180,E1 -15991.113,E2 -15991.113} C_VEL
LIN {X 0,Y 305.566,Z 417.418,A -85,B 0,C 180,E1 -15994.087,E2 -15994.087} C_VEL
LIN {X 0,Y 305.495,Z 417.431,A -85,B 0,C 180,E1 -15998.402,E2 -15998.402} C_VEL
LIN {X 0,Y 305.584,Z 417.415,A -85,B 0,C 180,E1 -16001.217,E2 -16001.217} C_VEL
LIN {X 0,Y 305.631,Z 417.409,A -85,B 0,C 180,E1 -16005.348,E2 -16005.348} C_VEL
LIN {X 0,Y 305.631,Z 417.411,A -85,B 0,C 180,E1 -16009.399,E2 -16009.399} C_VEL
LIN {X 0,Y 305.808,Z 417.391,A -85,B 0,C 180,E1 -16012.074,E2 -16012.074} C_VEL
LIN {X 0,Y 305.685,Z 417.402,A -85,B 0,C 180,E1 -16014.723,E2 -16014.723} C_VEL
LIN {X 0,Y 305.952,Z 417.371,A -85,B 0,C 180,E1 -16018.684,E2 -16018.684} C_VEL
LIN {X 0,Y 305.952,Z 417.37,A -85,B 0,C 180,E1 -16021.316,E2 -16021.316} C_VEL
LIN {X 0,Y 305.845,Z 417.385,A -85,B 0,C 180,E1 -16026.597,E2 -16026.597} C_VEL
LIN {X 0,Y 305.729,Z 417.395,A -85,B 0,C 180,E1 -16029.26,E2 -16029.26} C_VEL
LIN {X 0,Y 305.582,Z 417.413,A -85,B 0,C 180,E1 -16033.296,E2 -16033.296} C_VEL
LIN {X 0,Y 305.587,Z 417.42,A -85,B 0,C 180,E1 -16036.02,E2 -16036.02} C_VEL
LIN {X 0,Y 305.57,Z 417.42,A -85,B 0,C 180,E1 -16039.445,E2 -16039.445} C_VEL
LIN {X 0,Y 305.483,Z 417.429,A -85,B 0,C 180,E1 -16043.041,E2 -16043.041} C_VEL
LIN {X 0,Y 305.541,Z 417.425,A -85,B 0,C 180,E1 -16046.227,E2 -16046.227} C_VEL
LIN {X 0,Y 305.49,Z 417.427,A -85,B 0,C 180,E1 -16049.05,E2 -16049.05} C_VEL
LIN {X 0,Y 305.442,Z 417.439,A -85,B 0,C 180,E1 -16051.952,E2 -16051.952} C_VEL
LIN {X 0,Y 305.457,Z 417.433,A -85,B 0,C 180,E1 -16055.114,E2 -16055.114} C_VEL
LIN {X 0,Y 305.489,Z 417.429,A -85,B 0,C 180,E1 -16058.54,E2 -16058.54} C_VEL
LIN {X 0,Y 305.517,Z 417.425,A -85,B 0,C 180,E1 -16062.6,E2 -16062.6} C_VEL
LIN {X 0,Y 305.53,Z 417.424,A -85,B 0,C 180,E1 -16066.365,E2 -16066.365} C_VEL
LIN {X 0,Y 305.481,Z 417.432,A -85,B 0,C 180,E1 -16069.897,E2 -16069.897} C_VEL
LIN {X 0,Y 305.499,Z 417.431,A -85,B 0,C 180,E1 -16073.627,E2 -16073.627} C_VEL
LIN {X 0,Y 305.462,Z 417.433,A -85,B 0,C 180,E1 -16076.484,E2 -16076.484} C_VEL
LIN {X 0,Y 305.494,Z 417.431,A -85,B 0,C 180,E1 -16080.951,E2 -16080.951} C_VEL
LIN {X 0,Y 305.57,Z 417.419,A -85,B 0,C 180,E1 -16084.089,E2 -16084.089} C_VEL
LIN {X 0,Y 305.404,Z 417.441,A -85,B 0,C 180,E1 -16088.396,E2 -16088.396} C_VEL
LIN {X 0,Y 305.402,Z 417.533,A -85,B 0,C 180,E1 -16089.104,E2 -16089.104} C_VEL
LIN {X 0,Y 305.088,Z 421.045,A -85,B 0,C 180,E1 -16092.575,E2 -16092.575} C_VEL
LIN {X 0,Y 304.984,Z 423.995,A -85,B 0,C 180,E1 -16095.429,E2 -16095.429} C_VEL
LIN {X 0,Y 304.681,Z 428.193,A -85,B 0,C 180,E1 -16099.367,E2 -16099.367} C_VEL
LIN {X 0,Y 304.624,Z 430.815,A -85,B 0,C 180,E1 -16101.801,E2 -16101.801} C_VEL
LIN {X 0,Y 307.749,Z 444.665,A -85,B 0,C 180,E1 -16102.632,E2 -16102.632} C_VEL
LIN {X 0,Y 309.771,Z 455.842,A -85,B 0,C 180,E1 -16103.487,E2 -16103.487} C_VEL
LIN {X 0,Y 311.204,Z 466.589,A -85,B 0,C 180,E1 -16104.493,E2 -16104.493} C_VEL
LIN {X 0,Y 310.15,Z 477.169,A -85,B 0,C 180,E1 -16105.59,E2 -16105.59} C_VEL
LIN {X 0,Y 308.997,Z 487.325,A -85,B 0,C 180,E1 -16106.904,E2 -16106.904} C_VEL
LIN {X 0,Y 307.802,Z 496.481,A -85,B 0,C 180,E1 -16108.365,E2 -16108.365} C_VEL
LIN {X 0,Y 306.706,Z 504.85,A -85,B 0,C 180,E1 -16110,E2 -16110} C_VEL
LIN {X 0,Y 305.578,Z 513.048,A -85,B 0,C 180,E1 -16111.977,E2 -16111.977} C_VEL
LIN {X 0,Y 304.826,Z 519.632,A -85,B 0,C 180,E1 -16113.966,E2 -16113.966} C_VEL
LIN {X 0,Y 304.345,Z 524.773,A -85,B 0,C 180,E1 -16115.923,E2 -16115.923} C_VEL
LIN {X 0,Y 303.914,Z 528.959,A -85,B 0,C 180,E1 -16117.976,E2 -16117.976} C_VEL
LIN {X 0,Y 303.68,Z 531.077,A -85,B 0,C 180,E1 -16119.323,E2 -16119.323} C_VEL
LIN {X 0,Y 303.512,Z 532.757,A -85,B 0,C 180,E1 -16120.675,E2 -16120.675} C_VEL
LIN {X 0,Y 303.463,Z 534.025,A -85,B 0,C 180,E1 -16122.031,E2 -16122.031} C_VEL
LIN {X 0,Y 303.464,Z 534.876,A -85,B 0,C 180,E1 -16123.422,E2 -16123.422} C_VEL
LIN {X 0,Y 303.423,Z 535.27,A -85,B 0,C 180,E1 -16124.761,E2 -16124.761} C_VEL
LIN {X 0,Y 303.445,Z 535.278,A -85,B 0,C 180,E1 -16126.137,E2 -16126.137} C_VEL
LIN {X 0,Y 303.752,Z 534.348,A -85,B 0,C 180,E1 -16128.446,E2 -16128.446} C_VEL
LIN {X 0,Y 304.088,Z 532.73,A -85,B 0,C 180,E1 -16130.284,E2 -16130.284} C_VEL
LIN {X 0,Y 304.839,Z 529.343,A -85,B 0,C 180,E1 -16132.752,E2 -16132.752} C_VEL
LIN {X 0,Y 305.879,Z 524.484,A -85,B 0,C 180,E1 -16135.154,E2 -16135.154} C_VEL
LIN {X 0,Y 307.08,Z 518.887,A -85,B 0,C 180,E1 -16137.24,E2 -16137.24} C_VEL
LIN {X 0,Y 308.649,Z 511.807,A -85,B 0,C 180,E1 -16139.311,E2 -16139.311} C_VEL
LIN {X 0,Y 310.175,Z 504.384,A -85,B 0,C 180,E1 -16141.055,E2 -16141.055} C_VEL
LIN {X 0,Y 311.963,Z 495.543,A -85,B 0,C 180,E1 -16142.729,E2 -16142.729} C_VEL
LIN {X 0,Y 313.832,Z 485.622,A -85,B 0,C 180,E1 -16144.239,E2 -16144.239} C_VEL
LIN {X 0,Y 315.526,Z 474.955,A -85,B 0,C 180,E1 -16145.546,E2 -16145.546} C_VEL
LIN {X 0,Y 315.924,Z 471.022,A -85,B 0,C 180,E1 -16145.97,E2 -16145.97} C_VEL
LIN {X 0,Y 314.205,Z 461.031,A -85,B 0,C 180,E1 -16147.151,E2 -16147.151} C_VEL
LIN {X 0,Y 311.022,Z 448.798,A -85,B 0,C 180,E1 -16148.447,E2 -16148.447} C_VEL
LIN {X 0,Y 306.792,Z 436.512,A -85,B 0,C 180,E1 -16149.593,E2 -16149.593} C_VEL
LIN {X 0,Y 305.077,Z 431.68,A -85,B 0,C 180,E1 -16149.985,E2 -16149.985} C_VEL
LIN {X 0,Y 305.036,Z 431.271,A -85,B 0,C 180,E1 -16150.174,E2 -16150.174} C_VEL
LIN {X 0,Y 305.378,Z 427.924,A -85,B 0,C 180,E1 -16153.663,E2 -16153.663} C_VEL
LIN {X 0,Y 305.743,Z 424.533,A -85,B 0,C 180,E1 -16157.355,E2 -16157.355} C_VEL
LIN {X 0,Y 305.887,Z 422.267,A -85,B 0,C 180,E1 -16159.96,E2 -16159.96} C_VEL
LIN {X 0,Y 305.714,Z 419.313,A -85,B 0,C 180,E1 -16163.571,E2 -16163.571} C_VEL
LIN {X 0,Y 305.497,Z 417.529,A -85,B 0,C 180,E1 -16165.911,E2 -16165.911} C_VEL
LIN {X 0,Y 305.462,Z 417.437,A -85,B 0,C 180,E1 -16169.591,E2 -16169.591} C_VEL
LIN {X 0,Y 305.517,Z 417.429,A -85,B 0,C 180,E1 -16172.608,E2 -16172.608} C_VEL
LIN {X 0,Y 305.5,Z 417.431,A -85,B 0,C 180,E1 -16175.538,E2 -16175.538} C_VEL
LIN {X 0,Y 305.508,Z 417.43,A -85,B 0,C 180,E1 -16179.814,E2 -16179.814} C_VEL
LIN {X 0,Y 305.57,Z 417.42,A -85,B 0,C 180,E1 -16182.603,E2 -16182.603} C_VEL
LIN {X 0,Y 305.644,Z 417.411,A -85,B 0,C 180,E1 -16185.349,E2 -16185.349} C_VEL
LIN {X 0,Y 305.582,Z 417.418,A -85,B 0,C 180,E1 -16186.535,E2 -16186.535} C_VEL
LIN {X 0,Y 304.941,Z 417.504,A -85,B 0,C 180,E1 -16187.635,E2 -16187.635} C_VEL
LIN {X 0,Y 302.167,Z 417.851,A -85,B 0,C 180,E1 -16189.43,E2 -16189.43} C_VEL
LIN {X 0,Y 299.819,Z 418.14,A -85,B 0,C 180,E1 -16190.885,E2 -16190.885} C_VEL
LIN {X 0,Y 298.823,Z 418.263,A -85,B 0,C 180,E1 -16192.01,E2 -16192.01} C_VEL
LIN {X 0,Y 298.749,Z 418.27,A -85,B 0,C 180,E1 -16192.391,E2 -16192.391} C_VEL
LIN {X 0,Y 298.832,Z 418.26,A -85,B 0,C 180,E1 -16197.304,E2 -16197.304} C_VEL
LIN {X 0,Y 299.005,Z 418.241,A -85,B 0,C 180,E1 -16200,E2 -16200} C_VEL
LIN {X 0,Y 298.833,Z 418.261,A -85,B 0,C 180,E1 -16202.696,E2 -16202.696} C_VEL
LIN {X 0,Y 298.789,Z 418.263,A -85,B 0,C 180,E1 -16206.754,E2 -16206.754} C_VEL
LIN {X 0,Y 298.677,Z 418.282,A -85,B 0,C 180,E1 -16209.481,E2 -16209.481} C_VEL
LIN {X 0,Y 298.55,Z 418.296,A -85,B 0,C 180,E1 -16213.616,E2 -16213.616} C_VEL
LIN {X 0,Y 298.546,Z 418.3,A -85,B 0,C 180,E1 -16216.409,E2 -16216.409} C_VEL
LIN {X 0,Y 298.508,Z 418.305,A -85,B 0,C 180,E1 -16219.655,E2 -16219.655} C_VEL
LIN {X 0,Y 298.454,Z 418.312,A -85,B 0,C 180,E1 -16223.598,E2 -16223.598} C_VEL
LIN {X 0,Y 298.487,Z 418.307,A -85,B 0,C 180,E1 -16226.575,E2 -16226.575} C_VEL
LIN {X 0,Y 298.419,Z 418.314,A -85,B 0,C 180,E1 -16229.642,E2 -16229.642} C_VEL
LIN {X 0,Y 298.393,Z 418.317,A -85,B 0,C 180,E1 -16232.801,E2 -16232.801} C_VEL
LIN {X 0,Y 298.442,Z 418.306,A -85,B 0,C 180,E1 -16236.808,E2 -16236.808} C_VEL
LIN {X 0,Y 298.43,Z 418.333,A -85,B 0,C 180,E1 -16239.181,E2 -16239.181} C_VEL
LIN {X 0,Y 298.998,Z 421.94,A -85,B 0,C 180,E1 -16243.227,E2 -16243.227} C_VEL
LIN {X 0,Y 299.701,Z 425.771,A -85,B 0,C 180,E1 -16247.153,E2 -16247.153} C_VEL
LIN {X 0,Y 300.256,Z 429.658,A -85,B 0,C 180,E1 -16250.804,E2 -16250.804} C_VEL
LIN {X 0,Y 300.473,Z 431.792,A -85,B 0,C 180,E1 -16252.68,E2 -16252.68} C_VEL
LIN {X 0,Y 300.207,Z 435.604,A -85,B 0,C 180,E1 -16255.817,E2 -16255.817} C_VEL
LIN {X 0,Y 299.545,Z 439.607,A -85,B 0,C 180,E1 -16258.925,E2 -16258.925} C_VEL
LIN {X 0,Y 298.657,Z 445.198,A -85,B 0,C 180,E1 -16263.103,E2 -16263.103} C_VEL
LIN {X 0,Y 298.604,Z 445.455,A -85,B 0,C 180,E1 -16263.289,E2 -16263.289} C_VEL
LIN {X 0,Y 300.584,Z 452.009,A -85,B 0,C 180,E1 -16263.798,E2 -16263.798} C_VEL
LIN {X 0,Y 303.768,Z 463.218,A -85,B 0,C 180,E1 -16264.783,E2 -16264.783} C_VEL
LIN {X 0,Y 305.892,Z 473.344,A -85,B 0,C 180,E1 -16265.777,E2 -16265.777} C_VEL
LIN {X 0,Y 307.473,Z 485.599,A -85,B 0,C 180,E1 -16267.134,E2 -16267.134} C_VEL
LIN {X 0,Y 307.755,Z 494.306,A -85,B 0,C 180,E1 -16268.217,E2 -16268.217} C_VEL
LIN {X 0,Y 305.719,Z 505.185,A -85,B 0,C 180,E1 -16269.653,E2 -16269.653} C_VEL
LIN {X 0,Y 303.659,Z 515.296,A -85,B 0,C 180,E1 -16271.338,E2 -16271.338} C_VEL
LIN {X 0,Y 302,Z 523.711,A -85,B 0,C 180,E1 -16273.089,E2 -16273.089} C_VEL
LIN {X 0,Y 300.27,Z 531.462,A -85,B 0,C 180,E1 -16275.081,E2 -16275.081} C_VEL
LIN {X 0,Y 298.819,Z 537.69,A -85,B 0,C 180,E1 -16277.089,E2 -16277.089} C_VEL
LIN {X 0,Y 297.84,Z 542.667,A -85,B 0,C 180,E1 -16279.119,E2 -16279.119} C_VEL
LIN {X 0,Y 297.164,Z 546.538,A -85,B 0,C 180,E1 -16281.157,E2 -16281.157} C_VEL
LIN {X 0,Y 296.745,Z 549.404,A -85,B 0,C 180,E1 -16283.199,E2 -16283.199} C_VEL
LIN {X 0,Y 296.5,Z 551.748,A -85,B 0,C 180,E1 -16285.922,E2 -16285.922} C_VEL
LIN {X 0,Y 296.528,Z 552.344,A -85,B 0,C 180,E1 -16287.283,E2 -16287.283} C_VEL
LIN {X 0,Y 296.493,Z 552.527,A -85,B 0,C 180,E1 -16288.642,E2 -16288.642} C_VEL
LIN {X 0,Y 296.521,Z 552.294,A -85,B 0,C 180,E1 -16290,E2 -16290} C_VEL
LIN {X 0,Y 296.499,Z 551.672,A -85,B 0,C 180,E1 -16291.358,E2 -16291.358} C_VEL
LIN {X 0,Y 296.541,Z 550.66,A -85,B 0,C 180,E1 -16292.717,E2 -16292.717} C_VEL
LIN {X 0,Y 296.533,Z 549.218,A -85,B 0,C 180,E1 -16294.077,E2 -16294.077} C_VEL
LIN {X 0,Y 296.614,Z 546.227,A -85,B 0,C 180,E1 -16296.12,E2 -16296.12} C_VEL
LIN {X 0,Y 296.893,Z 542.167,A -85,B 0,C 180,E1 -16298.165,E2 -16298.165} C_VEL
LIN {X 0,Y 297.497,Z 535.908,A -85,B 0,C 180,E1 -16300.549,E2 -16300.549} C_VEL
LIN {X 0,Y 298.253,Z 529.074,A -85,B 0,C 180,E1 -16302.589,E2 -16302.589} C_VEL
LIN {X 0,Y 299.225,Z 522.107,A -85,B 0,C 180,E1 -16304.277,E2 -16304.277} C_VEL
LIN {X 0,Y 300.364,Z 513.7,A -85,B 0,C 180,E1 -16305.957,E2 -16305.957} C_VEL
LIN {X 0,Y 301.42,Z 504.437,A -85,B 0,C 180,E1 -16307.477,E2 -16307.477} C_VEL
LIN {X 0,Y 302.609,Z 494.476,A -85,B 0,C 180,E1 -16308.798,E2 -16308.798} C_VEL
LIN {X 0,Y 303.228,Z 488.541,A -85,B 0,C 180,E1 -16309.461,E2 -16309.461} C_VEL
LIN {X 0,Y 302.165,Z 476.334,A -85,B 0,C 180,E1 -16310.701,E2 -16310.701} C_VEL
LIN {X 0,Y 300.678,Z 464.313,A -85,B 0,C 180,E1 -16311.671,E2 -16311.671} C_VEL
LIN {X 0,Y 298.451,Z 450.817,A -85,B 0,C 180,E1 -16312.492,E2 -16312.492} C_VEL
LIN {X 0,Y 297.558,Z 446.071,A -85,B 0,C 180,E1 -16312.739,E2 -16312.739} C_VEL
LIN {X 0,Y 298.117,Z 440.408,A -85,B 0,C 180,E1 -16316.609,E2 -16316.609} C_VEL
LIN {X 0,Y 298.908,Z 433.91,A -85,B 0,C 180,E1 -16321.148,E2 -16321.148} C_VEL
LIN {X 0,Y 299.582,Z 428.828,A -85,B 0,C 180,E1 -16324.807,E2 -16324.807} C_VEL
LIN {X 0,Y 299.665,Z 425.134,A -85,B 0,C 180,E1 -16327.572,E2 -16327.572} C_VEL
LIN {X 0,Y 298.891,Z 420.641,A -85,B 0,C 180,E1 -16331.198,E2 -16331.198} C_VEL
LIN {X 0,Y 298.492,Z 418.306,A -85,B 0,C 180,E1 -16333.269,E2 -16333.269} C_VEL
LIN {X 0,Y 298.429,Z 418.314,A -85,B 0,C 180,E1 -16336.925,E2 -16336.925} C_VEL
LIN {X 0,Y 298.4,Z 418.318,A -85,B 0,C 180,E1 -16341.005,E2 -16341.005} C_VEL
LIN {X 0,Y 298.414,Z 418.311,A -85,B 0,C 180,E1 -16343.929,E2 -16343.929} C_VEL
LIN {X 0,Y 298.391,Z 418.314,A -85,B 0,C 180,E1 -16347.983,E2 -16347.983} C_VEL
LIN {X 0,Y 298.459,Z 418.301,A -85,B 0,C 180,E1 -16351.904,E2 -16351.904} C_VEL
LIN {X 0,Y 298.48,Z 418.306,A -85,B 0,C 180,E1 -16354.923,E2 -16354.923} C_VEL
LIN {X 0,Y 298.445,Z 418.306,A -85,B 0,C 180,E1 -16359.315,E2 -16359.315} C_VEL
LIN {X 0,Y 298.53,Z 418.294,A -85,B 0,C 180,E1 -16362.179,E2 -16362.179} C_VEL
LIN {X 0,Y 298.579,Z 418.288,A -85,B 0,C 180,E1 -16364.994,E2 -16364.994} C_VEL
LIN {X 0,Y 298.586,Z 418.29,A -85,B 0,C 180,E1 -16369.146,E2 -16369.146} C_VEL
LIN {X 0,Y 298.754,Z 418.268,A -85,B 0,C 180,E1 -16371.886,E2 -16371.886} C_VEL
LIN {X 0,Y 298.656,Z 418.278,A -85,B 0,C 180,E1 -16374.599,E2 -16374.599} C_VEL
LIN {X 0,Y 298.918,Z 418.247,A -85,B 0,C 180,E1 -16378.653,E2 -16378.653} C_VEL
LIN {X 0,Y 298.918,Z 418.246,A -85,B 0,C 180,E1 -16381.347,E2 -16381.347} C_VEL
LIN {X 0,Y 298.791,Z 418.263,A -85,B 0,C 180,E1 -16386.754,E2 -16386.754} C_VEL
LIN {X 0,Y 298.674,Z 418.274,A -85,B 0,C 180,E1 -16389.48,E2 -16389.48} C_VEL
LIN {X 0,Y 298.545,Z 418.29,A -85,B 0,C 180,E1 -16393.615,E2 -16393.615} C_VEL
LIN {X 0,Y 298.542,Z 418.297,A -85,B 0,C 180,E1 -16396.409,E2 -16396.409} C_VEL
LIN {X 0,Y 298.505,Z 418.302,A -85,B 0,C 180,E1 -16399.655,E2 -16399.655} C_VEL
LIN {X 0,Y 298.451,Z 418.307,A -85,B 0,C 180,E1 -16403.598,E2 -16403.598} C_VEL
LIN {X 0,Y 298.483,Z 418.302,A -85,B 0,C 180,E1 -16406.575,E2 -16406.575} C_VEL
LIN {X 0,Y 298.416,Z 418.312,A -85,B 0,C 180,E1 -16409.641,E2 -16409.641} C_VEL
LIN {X 0,Y 298.392,Z 418.313,A -85,B 0,C 180,E1 -16412.8,E2 -16412.8} C_VEL
